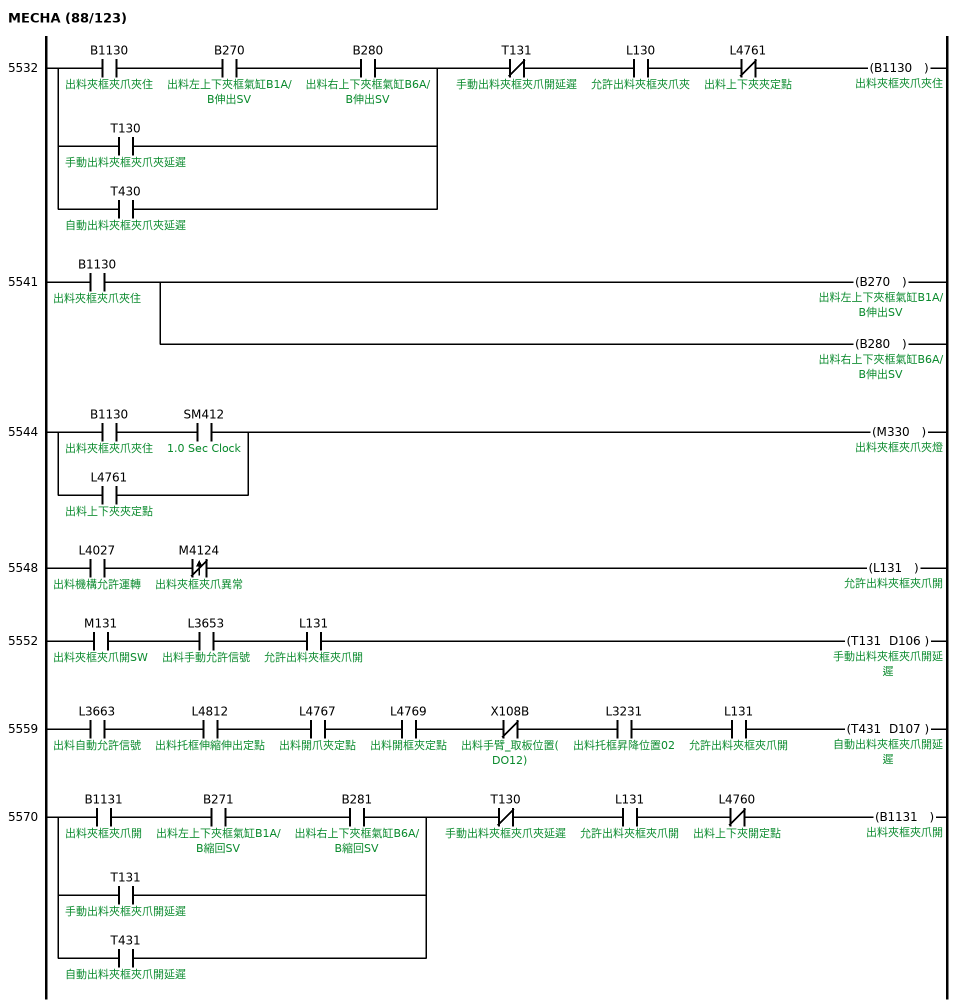
[picture p384: ladder of MECHA, rungs at steps 5532 to 5570]
5532  LD      B1130  ; 出料夾框夾爪夾住
      AND     B270  ; 出料左上下夾框氣缸B1A/B伸出SV
      AND     B280  ; 出料右上下夾框氣缸B6A/B伸出SV
      OR      T130  ; 手動出料夾框夾爪夾延遲
      OR      T430  ; 自動出料夾框夾爪夾延遲
      ANI     T131  ; 手動出料夾框夾爪開延遲
      AND     L130  ; 允許出料夾框夾爪夾
      ANI     L4761  ; 出料上下夾夾定點
      OUT     B1130  ; 出料夾框夾爪夾住
5541  LD      B1130  ; 出料夾框夾爪夾住
      OUT     B270  ; 出料左上下夾框氣缸B1A/B伸出SV
      OUT     B280  ; 出料右上下夾框氣缸B6A/B伸出SV
5544  LD      B1130  ; 出料夾框夾爪夾住
      AND     SM412  ; 1.0 Sec Clock
      OR      L4761  ; 出料上下夾夾定點
      OUT     M330  ; 出料夾框夾爪夾燈
5548  LD      L4027  ; 出料機構允許運轉
      ANDPI   M4124  ; 出料夾框夾爪異常
      OUT     L131  ; 允許出料夾框夾爪開
5552  LD      M131  ; 出料夾框夾爪開SW
      AND     L3653  ; 出料手動允許信號
      AND     L131  ; 允許出料夾框夾爪開
      OUT     T131 D106  ; 手動出料夾框夾爪開延遲
5559  LD      L3663  ; 出料自動允許信號
      AND     L4812  ; 出料托框伸縮伸出定點
      AND     L4767  ; 出料開爪夾定點
      AND     L4769  ; 出料開框夾定點
      ANI     X108B  ; 出料手臂_取板位置(DO12)
      AND     L3231  ; 出料托框昇降位置02
      AND     L131  ; 允許出料夾框夾爪開
      OUT     T431 D107  ; 自動出料夾框夾爪開延遲
5570  LD      B1131  ; 出料夾框夾爪開
      AND     B271  ; 出料左上下夾框氣缸B1A/B縮回SV
      AND     B281  ; 出料右上下夾框氣缸B6A/B縮回SV
      OR      T131  ; 手動出料夾框夾爪開延遲
      OR      T431  ; 自動出料夾框夾爪開延遲
      ANI     T130  ; 手動出料夾框夾爪夾延遲
      AND     L131  ; 允許出料夾框夾爪開
      ANI     L4760  ; 出料上下夾開定點
      OUT     B1131  ; 出料夾框夾爪開
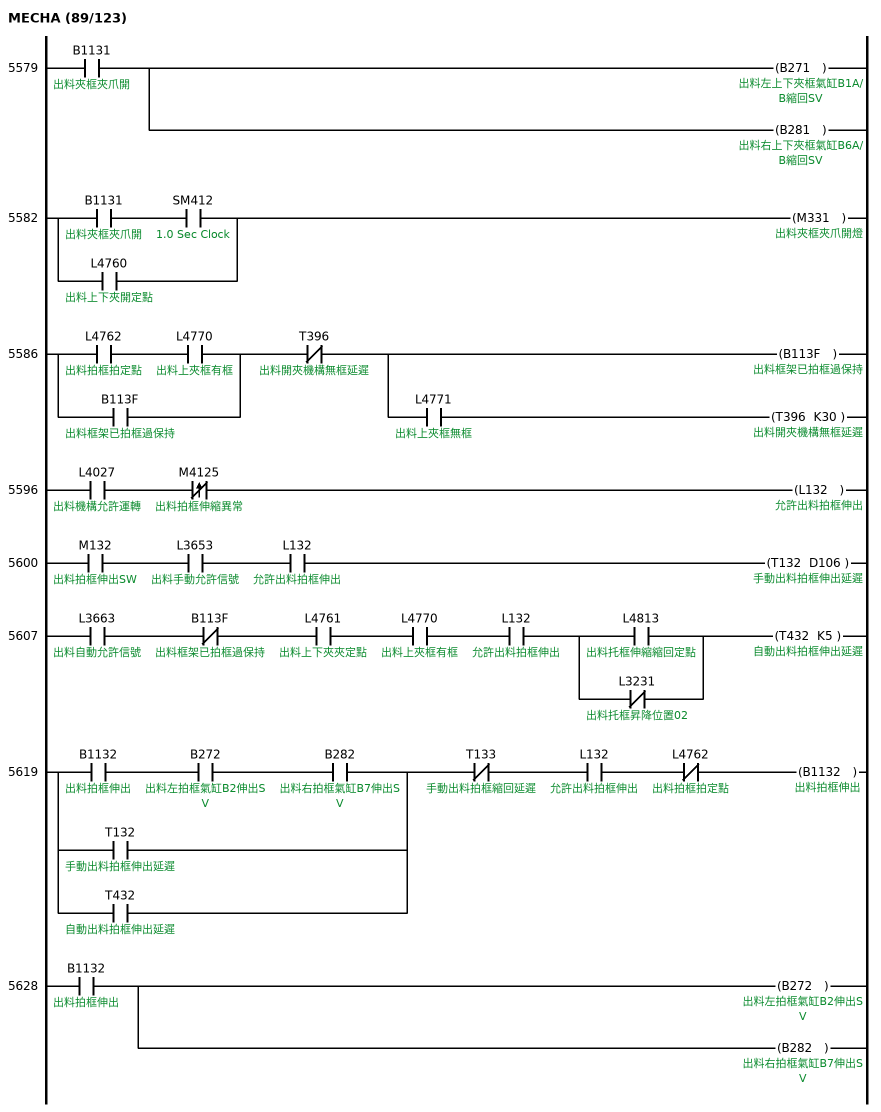
5579  LD      B1131  ; 出料夾框夾爪開
      OUT     B271  ; 出料左上下夾框氣缸B1A/B縮回SV
      OUT     B281  ; 出料右上下夾框氣缸B6A/B縮回SV
5582  LD      B1131  ; 出料夾框夾爪開
      AND     SM412  ; 1.0 Sec Clock
      OR      L4760  ; 出料上下夾開定點
      OUT     M331  ; 出料夾框夾爪開燈
5586  LD      L4762  ; 出料拍框拍定點
      AND     L4770  ; 出料上夾框有框
      OR      B113F  ; 出料框架已拍框過保持
      ANI     T396  ; 出料開夾機構無框延遲
      OUT     B113F  ; 出料框架已拍框過保持
      AND     L4771  ; 出料上夾框無框
      OUT     T396 K30  ; 出料開夾機構無框延遲
5596  LD      L4027  ; 出料機構允許運轉
      ANDPI   M4125  ; 出料拍框伸縮異常
      OUT     L132  ; 允許出料拍框伸出
5600  LD      M132  ; 出料拍框伸出SW
      AND     L3653  ; 出料手動允許信號
      AND     L132  ; 允許出料拍框伸出
      OUT     T132 D106  ; 手動出料拍框伸出延遲
5607  LD      L3663  ; 出料自動允許信號
      ANI     B113F  ; 出料框架已拍框過保持
      AND     L4761  ; 出料上下夾夾定點
      AND     L4770  ; 出料上夾框有框
      AND     L132  ; 允許出料拍框伸出
      LD      L4813  ; 出料托框伸縮縮回定點
      ORI     L3231  ; 出料托框昇降位置02
      ANB
      OUT     T432 K5  ; 自動出料拍框伸出延遲
5619  LD      B1132  ; 出料拍框伸出
      AND     B272  ; 出料左拍框氣缸B2伸出SV
      AND     B282  ; 出料右拍框氣缸B7伸出SV
      OR      T132  ; 手動出料拍框伸出延遲
      OR      T432  ; 自動出料拍框伸出延遲
      ANI     T133  ; 手動出料拍框縮回延遲
      AND     L132  ; 允許出料拍框伸出
      ANI     L4762  ; 出料拍框拍定點
      OUT     B1132  ; 出料拍框伸出
5628  LD      B1132  ; 出料拍框伸出
      OUT     B272  ; 出料左拍框氣缸B2伸出SV
      OUT     B282  ; 出料右拍框氣缸B7伸出SV
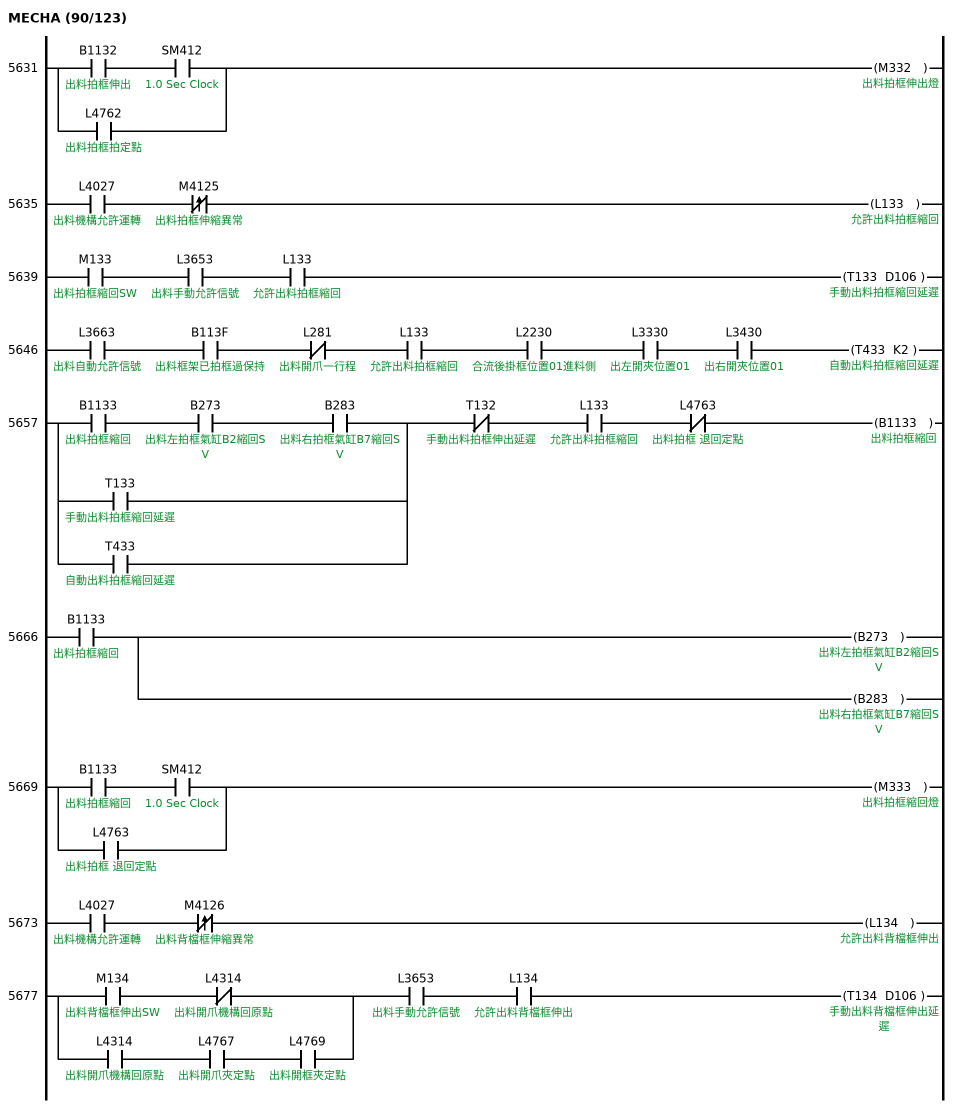
5631  LD      B1132  ; 出料拍框伸出
      AND     SM412  ; 1.0 Sec Clock
      OR      L4762  ; 出料拍框拍定點
      OUT     M332  ; 出料拍框伸出燈
5635  LD      L4027  ; 出料機構允許運轉
      ANDPI   M4125  ; 出料拍框伸縮異常
      OUT     L133  ; 允許出料拍框縮回
5639  LD      M133  ; 出料拍框縮回SW
      AND     L3653  ; 出料手動允許信號
      AND     L133  ; 允許出料拍框縮回
      OUT     T133 D106  ; 手動出料拍框縮回延遲
5646  LD      L3663  ; 出料自動允許信號
      AND     B113F  ; 出料框架已拍框過保持
      ANI     L281  ; 出料開爪一行程
      AND     L133  ; 允許出料拍框縮回
      AND     L2230  ; 合流後掛框位置01進料側
      AND     L3330  ; 出左開夾位置01
      AND     L3430  ; 出右開夾位置01
      OUT     T433 K2  ; 自動出料拍框縮回延遲
5657  LD      B1133  ; 出料拍框縮回
      AND     B273  ; 出料左拍框氣缸B2縮回SV
      AND     B283  ; 出料右拍框氣缸B7縮回SV
      OR      T133  ; 手動出料拍框縮回延遲
      OR      T433  ; 自動出料拍框縮回延遲
      ANI     T132  ; 手動出料拍框伸出延遲
      AND     L133  ; 允許出料拍框縮回
      ANI     L4763  ; 出料拍框 退回定點
      OUT     B1133  ; 出料拍框縮回
5666  LD      B1133  ; 出料拍框縮回
      OUT     B273  ; 出料左拍框氣缸B2縮回SV
      OUT     B283  ; 出料右拍框氣缸B7縮回SV
5669  LD      B1133  ; 出料拍框縮回
      AND     SM412  ; 1.0 Sec Clock
      OR      L4763  ; 出料拍框 退回定點
      OUT     M333  ; 出料拍框縮回燈
5673  LD      L4027  ; 出料機構允許運轉
      ANDPI   M4126  ; 出料背檔框伸縮異常
      OUT     L134  ; 允許出料背檔框伸出
5677  LD      M134  ; 出料背檔框伸出SW
      ANI     L4314  ; 出料開爪機構回原點
      LD      L4314  ; 出料開爪機構回原點
      AND     L4767  ; 出料開爪夾定點
      AND     L4769  ; 出料開框夾定點
      ORB
      AND     L3653  ; 出料手動允許信號
      AND     L134  ; 允許出料背檔框伸出
      OUT     T134 D106  ; 手動出料背檔框伸出延遲
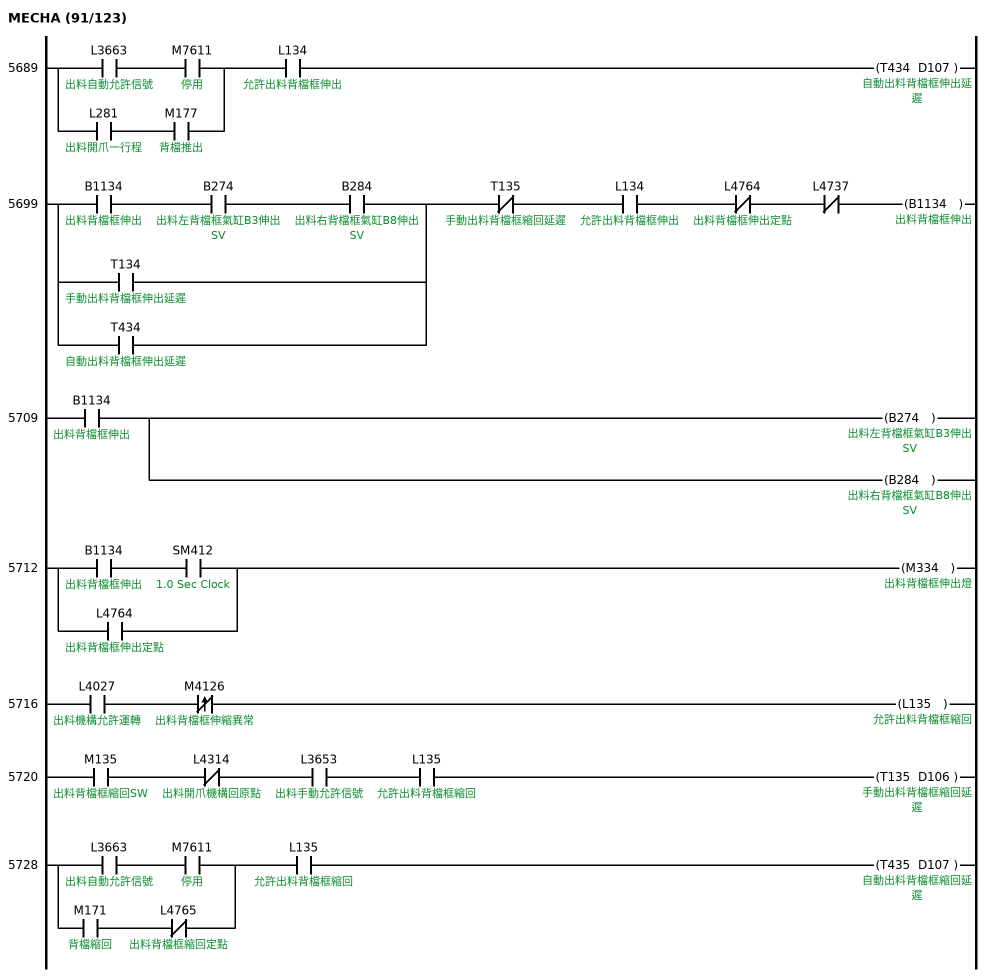
5689  LD      L3663  ; 出料自動允許信號
      AND     M7611  ; 停用
      LD      L281  ; 出料開爪一行程
      AND     M177  ; 背檔推出
      ORB
      AND     L134  ; 允許出料背檔框伸出
      OUT     T434 D107  ; 自動出料背檔框伸出延遲
5699  LD      B1134  ; 出料背檔框伸出
      AND     B274  ; 出料左背檔框氣缸B3伸出SV
      AND     B284  ; 出料右背檔框氣缸B8伸出SV
      OR      T134  ; 手動出料背檔框伸出延遲
      OR      T434  ; 自動出料背檔框伸出延遲
      ANI     T135  ; 手動出料背檔框縮回延遲
      AND     L134  ; 允許出料背檔框伸出
      ANI     L4764  ; 出料背檔框伸出定點
      ANI     L4737
      OUT     B1134  ; 出料背檔框伸出
5709  LD      B1134  ; 出料背檔框伸出
      OUT     B274  ; 出料左背檔框氣缸B3伸出SV
      OUT     B284  ; 出料右背檔框氣缸B8伸出SV
5712  LD      B1134  ; 出料背檔框伸出
      AND     SM412  ; 1.0 Sec Clock
      OR      L4764  ; 出料背檔框伸出定點
      OUT     M334  ; 出料背檔框伸出燈
5716  LD      L4027  ; 出料機構允許運轉
      ANDPI   M4126  ; 出料背檔框伸縮異常
      OUT     L135  ; 允許出料背檔框縮回
5720  LD      M135  ; 出料背檔框縮回SW
      ANI     L4314  ; 出料開爪機構回原點
      AND     L3653  ; 出料手動允許信號
      AND     L135  ; 允許出料背檔框縮回
      OUT     T135 D106  ; 手動出料背檔框縮回延遲
5728  LD      L3663  ; 出料自動允許信號
      AND     M7611  ; 停用
      LD      M171  ; 背檔縮回
      ANI     L4765  ; 出料背檔框縮回定點
      ORB
      AND     L135  ; 允許出料背檔框縮回
      OUT     T435 D107  ; 自動出料背檔框縮回延遲
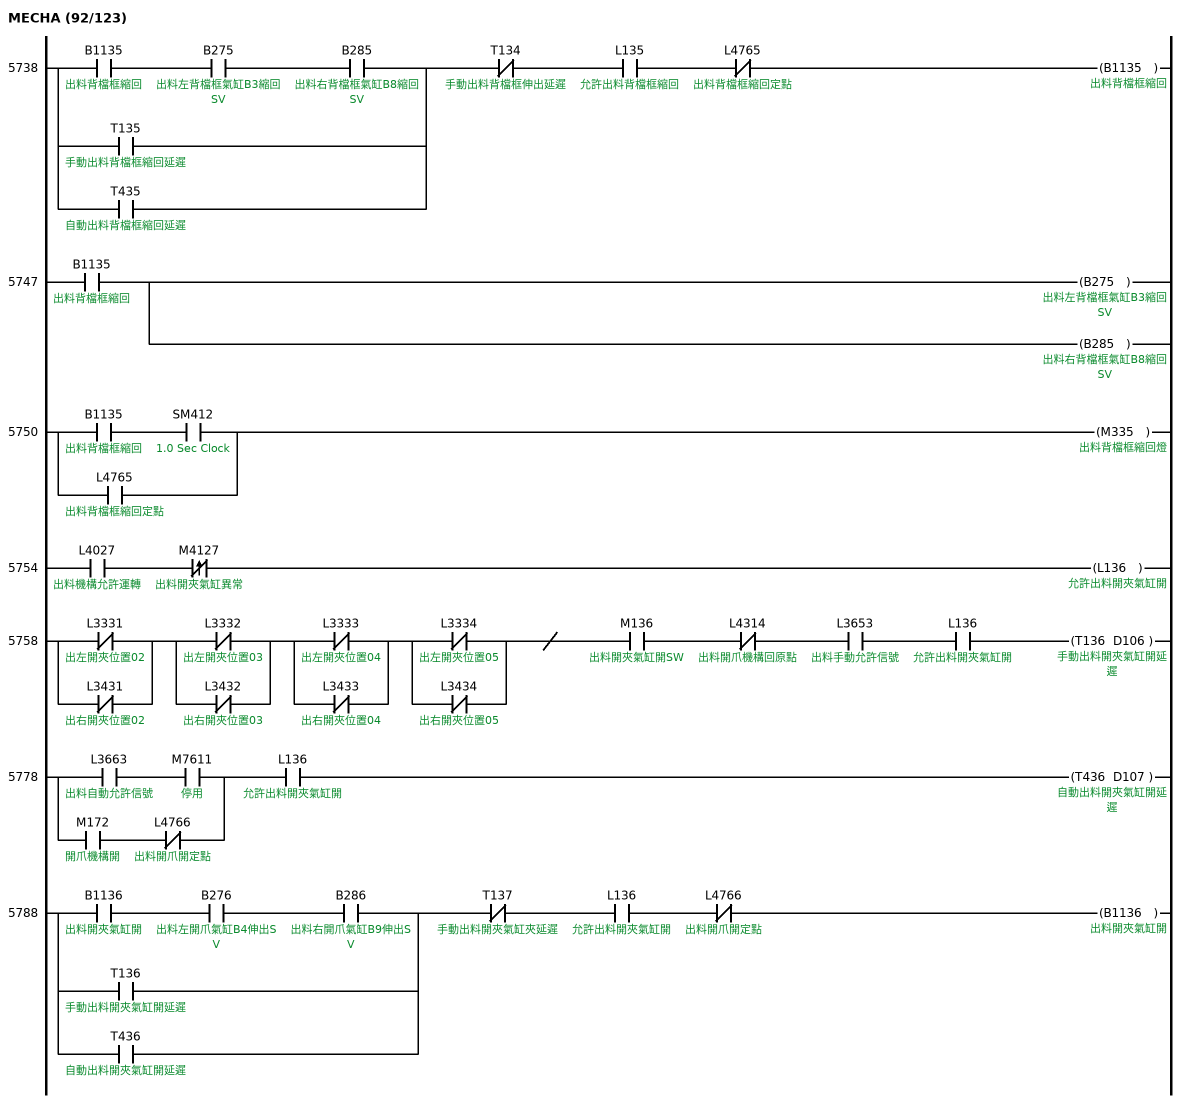
5738  LD      B1135  ; 出料背檔框縮回
      AND     B275  ; 出料左背檔框氣缸B3縮回SV
      AND     B285  ; 出料右背檔框氣缸B8縮回SV
      OR      T135  ; 手動出料背檔框縮回延遲
      OR      T435  ; 自動出料背檔框縮回延遲
      ANI     T134  ; 手動出料背檔框伸出延遲
      AND     L135  ; 允許出料背檔框縮回
      ANI     L4765  ; 出料背檔框縮回定點
      OUT     B1135  ; 出料背檔框縮回
5747  LD      B1135  ; 出料背檔框縮回
      OUT     B275  ; 出料左背檔框氣缸B3縮回SV
      OUT     B285  ; 出料右背檔框氣缸B8縮回SV
5750  LD      B1135  ; 出料背檔框縮回
      AND     SM412  ; 1.0 Sec Clock
      OR      L4765  ; 出料背檔框縮回定點
      OUT     M335  ; 出料背檔框縮回燈
5754  LD      L4027  ; 出料機構允許運轉
      ANDPI   M4127  ; 出料開夾氣缸異常
      OUT     L136  ; 允許出料開夾氣缸開
5758  LDI     L3331  ; 出左開夾位置02
      ORI     L3431  ; 出右開夾位置02
      LDI     L3332  ; 出左開夾位置03
      ORI     L3432  ; 出右開夾位置03
      ANB
      LDI     L3333  ; 出左開夾位置04
      ORI     L3433  ; 出右開夾位置04
      ANB
      LDI     L3334  ; 出左開夾位置05
      ORI     L3434  ; 出右開夾位置05
      ANB
      INV
      AND     M136  ; 出料開夾氣缸開SW
      ANI     L4314  ; 出料開爪機構回原點
      AND     L3653  ; 出料手動允許信號
      AND     L136  ; 允許出料開夾氣缸開
      OUT     T136 D106  ; 手動出料開夾氣缸開延遲
5778  LD      L3663  ; 出料自動允許信號
      AND     M7611  ; 停用
      LD      M172  ; 開爪機構開
      ANI     L4766  ; 出料開爪開定點
      ORB
      AND     L136  ; 允許出料開夾氣缸開
      OUT     T436 D107  ; 自動出料開夾氣缸開延遲
5788  LD      B1136  ; 出料開夾氣缸開
      AND     B276  ; 出料左開爪氣缸B4伸出SV
      AND     B286  ; 出料右開爪氣缸B9伸出SV
      OR      T136  ; 手動出料開夾氣缸開延遲
      OR      T436  ; 自動出料開夾氣缸開延遲
      ANI     T137  ; 手動出料開夾氣缸夾延遲
      AND     L136  ; 允許出料開夾氣缸開
      ANI     L4766  ; 出料開爪開定點
      OUT     B1136  ; 出料開夾氣缸開
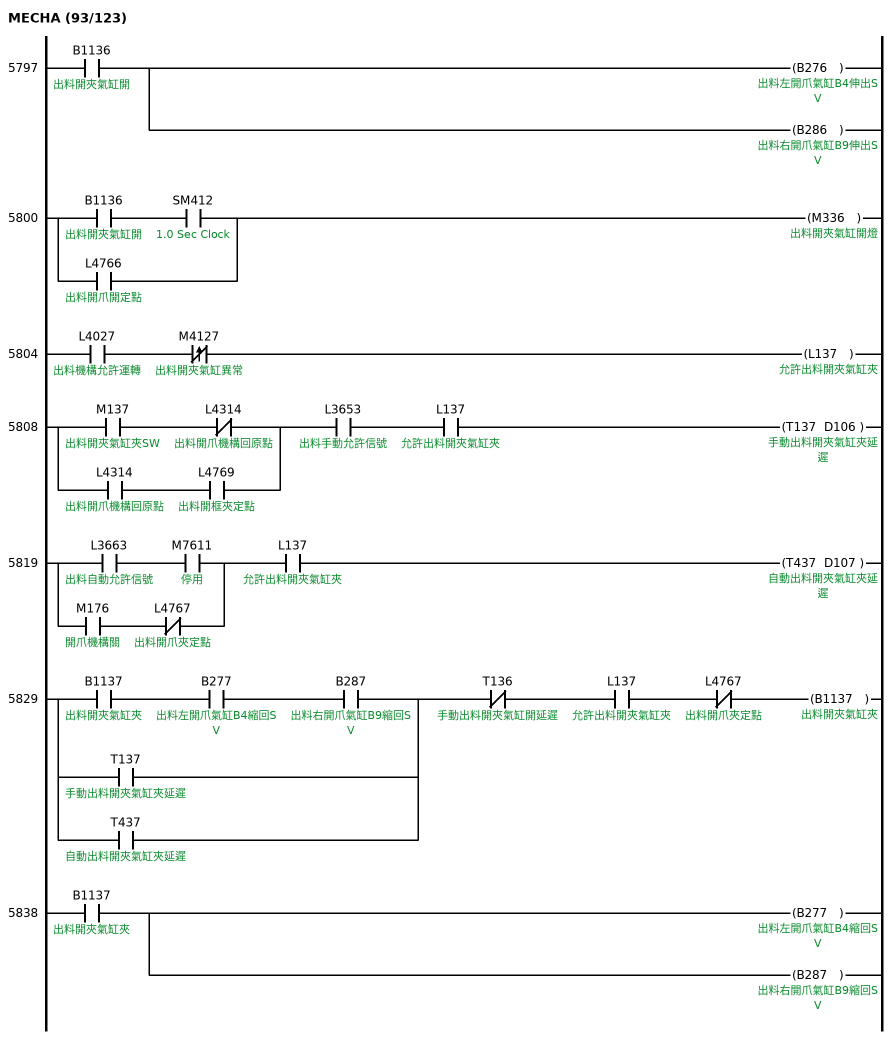
5797  LD      B1136  ; 出料開夾氣缸開
      OUT     B276  ; 出料左開爪氣缸B4伸出SV
      OUT     B286  ; 出料右開爪氣缸B9伸出SV
5800  LD      B1136  ; 出料開夾氣缸開
      AND     SM412  ; 1.0 Sec Clock
      OR      L4766  ; 出料開爪開定點
      OUT     M336  ; 出料開夾氣缸開燈
5804  LD      L4027  ; 出料機構允許運轉
      ANDPI   M4127  ; 出料開夾氣缸異常
      OUT     L137  ; 允許出料開夾氣缸夾
5808  LD      M137  ; 出料開夾氣缸夾SW
      ANI     L4314  ; 出料開爪機構回原點
      LD      L4314  ; 出料開爪機構回原點
      AND     L4769  ; 出料開框夾定點
      ORB
      AND     L3653  ; 出料手動允許信號
      AND     L137  ; 允許出料開夾氣缸夾
      OUT     T137 D106  ; 手動出料開夾氣缸夾延遲
5819  LD      L3663  ; 出料自動允許信號
      AND     M7611  ; 停用
      LD      M176  ; 開爪機構關
      ANI     L4767  ; 出料開爪夾定點
      ORB
      AND     L137  ; 允許出料開夾氣缸夾
      OUT     T437 D107  ; 自動出料開夾氣缸夾延遲
5829  LD      B1137  ; 出料開夾氣缸夾
      AND     B277  ; 出料左開爪氣缸B4縮回SV
      AND     B287  ; 出料右開爪氣缸B9縮回SV
      OR      T137  ; 手動出料開夾氣缸夾延遲
      OR      T437  ; 自動出料開夾氣缸夾延遲
      ANI     T136  ; 手動出料開夾氣缸開延遲
      AND     L137  ; 允許出料開夾氣缸夾
      ANI     L4767  ; 出料開爪夾定點
      OUT     B1137  ; 出料開夾氣缸夾
5838  LD      B1137  ; 出料開夾氣缸夾
      OUT     B277  ; 出料左開爪氣缸B4縮回SV
      OUT     B287  ; 出料右開爪氣缸B9縮回SV
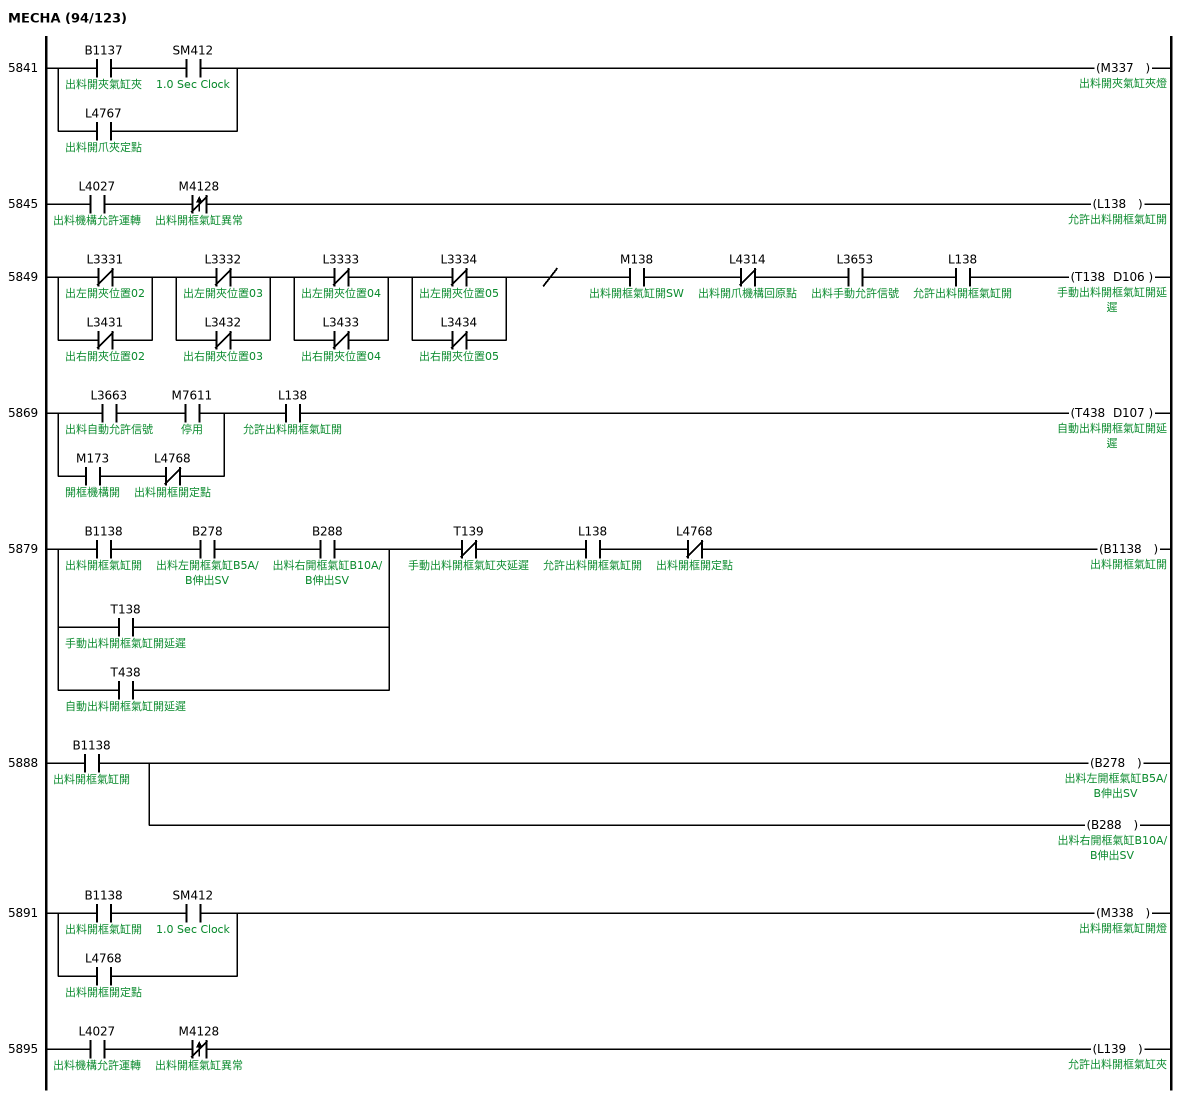
5841  LD      B1137  ; 出料開夾氣缸夾
      AND     SM412  ; 1.0 Sec Clock
      OR      L4767  ; 出料開爪夾定點
      OUT     M337  ; 出料開夾氣缸夾燈
5845  LD      L4027  ; 出料機構允許運轉
      ANDPI   M4128  ; 出料開框氣缸異常
      OUT     L138  ; 允許出料開框氣缸開
5849  LDI     L3331  ; 出左開夾位置02
      ORI     L3431  ; 出右開夾位置02
      LDI     L3332  ; 出左開夾位置03
      ORI     L3432  ; 出右開夾位置03
      ANB
      LDI     L3333  ; 出左開夾位置04
      ORI     L3433  ; 出右開夾位置04
      ANB
      LDI     L3334  ; 出左開夾位置05
      ORI     L3434  ; 出右開夾位置05
      ANB
      INV
      AND     M138  ; 出料開框氣缸開SW
      ANI     L4314  ; 出料開爪機構回原點
      AND     L3653  ; 出料手動允許信號
      AND     L138  ; 允許出料開框氣缸開
      OUT     T138 D106  ; 手動出料開框氣缸開延遲
5869  LD      L3663  ; 出料自動允許信號
      AND     M7611  ; 停用
      LD      M173  ; 開框機構開
      ANI     L4768  ; 出料開框開定點
      ORB
      AND     L138  ; 允許出料開框氣缸開
      OUT     T438 D107  ; 自動出料開框氣缸開延遲
5879  LD      B1138  ; 出料開框氣缸開
      AND     B278  ; 出料左開框氣缸B5A/B伸出SV
      AND     B288  ; 出料右開框氣缸B10A/B伸出SV
      OR      T138  ; 手動出料開框氣缸開延遲
      OR      T438  ; 自動出料開框氣缸開延遲
      ANI     T139  ; 手動出料開框氣缸夾延遲
      AND     L138  ; 允許出料開框氣缸開
      ANI     L4768  ; 出料開框開定點
      OUT     B1138  ; 出料開框氣缸開
5888  LD      B1138  ; 出料開框氣缸開
      OUT     B278  ; 出料左開框氣缸B5A/B伸出SV
      OUT     B288  ; 出料右開框氣缸B10A/B伸出SV
5891  LD      B1138  ; 出料開框氣缸開
      AND     SM412  ; 1.0 Sec Clock
      OR      L4768  ; 出料開框開定點
      OUT     M338  ; 出料開框氣缸開燈
5895  LD      L4027  ; 出料機構允許運轉
      ANDPI   M4128  ; 出料開框氣缸異常
      OUT     L139  ; 允許出料開框氣缸夾
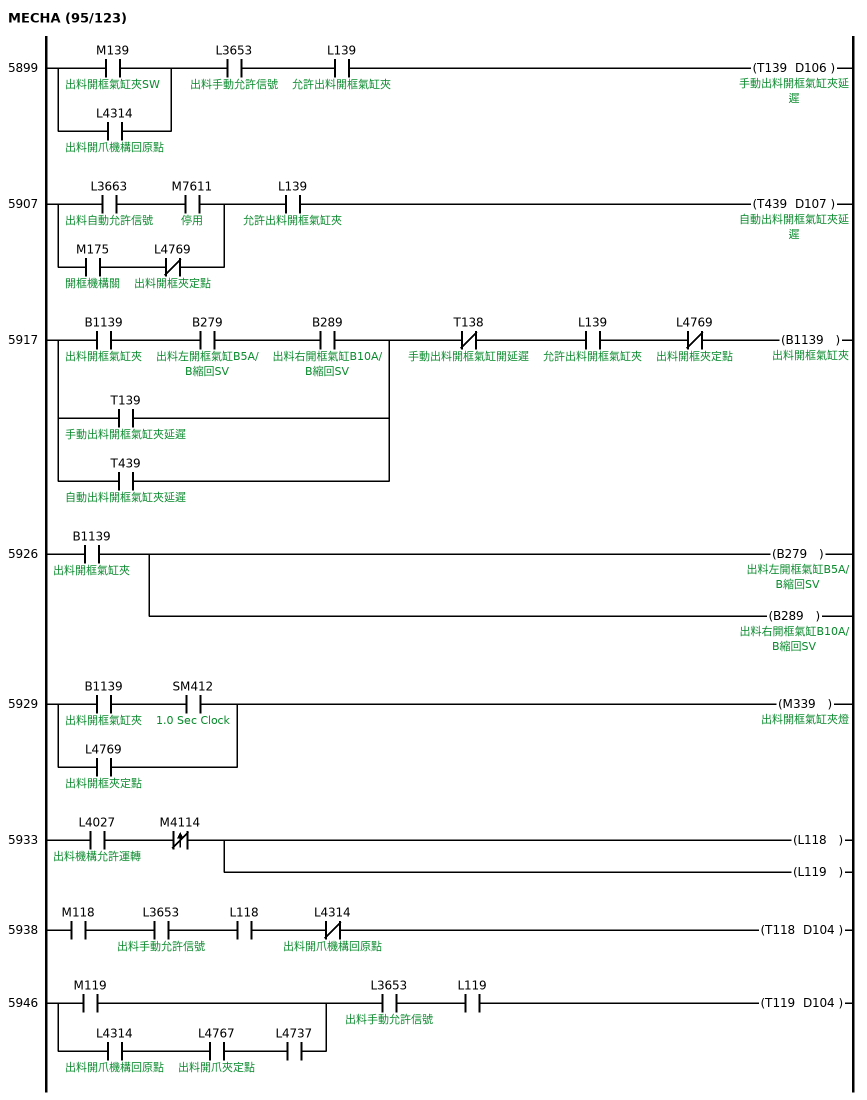
5899  LD      M139  ; 出料開框氣缸夾SW
      OR      L4314  ; 出料開爪機構回原點
      AND     L3653  ; 出料手動允許信號
      AND     L139  ; 允許出料開框氣缸夾
      OUT     T139 D106  ; 手動出料開框氣缸夾延遲
5907  LD      L3663  ; 出料自動允許信號
      AND     M7611  ; 停用
      LD      M175  ; 開框機構關
      ANI     L4769  ; 出料開框夾定點
      ORB
      AND     L139  ; 允許出料開框氣缸夾
      OUT     T439 D107  ; 自動出料開框氣缸夾延遲
5917  LD      B1139  ; 出料開框氣缸夾
      AND     B279  ; 出料左開框氣缸B5A/B縮回SV
      AND     B289  ; 出料右開框氣缸B10A/B縮回SV
      OR      T139  ; 手動出料開框氣缸夾延遲
      OR      T439  ; 自動出料開框氣缸夾延遲
      ANI     T138  ; 手動出料開框氣缸開延遲
      AND     L139  ; 允許出料開框氣缸夾
      ANI     L4769  ; 出料開框夾定點
      OUT     B1139  ; 出料開框氣缸夾
5926  LD      B1139  ; 出料開框氣缸夾
      OUT     B279  ; 出料左開框氣缸B5A/B縮回SV
      OUT     B289  ; 出料右開框氣缸B10A/B縮回SV
5929  LD      B1139  ; 出料開框氣缸夾
      AND     SM412  ; 1.0 Sec Clock
      OR      L4769  ; 出料開框夾定點
      OUT     M339  ; 出料開框氣缸夾燈
5933  LD      L4027  ; 出料機構允許運轉
      ANDPI   M4114
      OUT     L118
      OUT     L119
5938  LD      M118
      AND     L3653  ; 出料手動允許信號
      AND     L118
      ANI     L4314  ; 出料開爪機構回原點
      OUT     T118 D104
5946  LD      M119
      LD      L4314  ; 出料開爪機構回原點
      AND     L4767  ; 出料開爪夾定點
      AND     L4737
      ORB
      AND     L3653  ; 出料手動允許信號
      AND     L119
      OUT     T119 D104
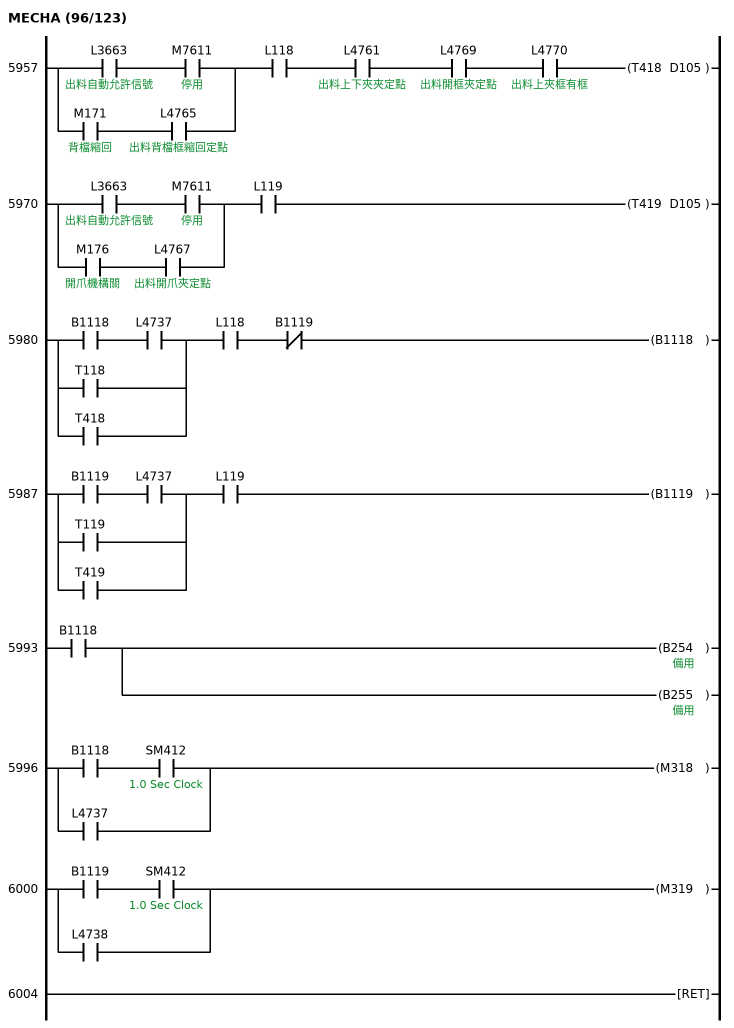
5957  LD      L3663  ; 出料自動允許信號
      AND     M7611  ; 停用
      LD      M171  ; 背檔縮回
      AND     L4765  ; 出料背檔框縮回定點
      ORB
      AND     L118
      AND     L4761  ; 出料上下夾夾定點
      AND     L4769  ; 出料開框夾定點
      AND     L4770  ; 出料上夾框有框
      OUT     T418 D105
5970  LD      L3663  ; 出料自動允許信號
      AND     M7611  ; 停用
      LD      M176  ; 開爪機構關
      AND     L4767  ; 出料開爪夾定點
      ORB
      AND     L119
      OUT     T419 D105
5980  LD      B1118
      AND     L4737
      OR      T118
      OR      T418
      AND     L118
      ANI     B1119
      OUT     B1118
5987  LD      B1119
      AND     L4737
      OR      T119
      OR      T419
      AND     L119
      OUT     B1119
5993  LD      B1118
      OUT     B254  ; 備用
      OUT     B255  ; 備用
5996  LD      B1118
      AND     SM412  ; 1.0 Sec Clock
      OR      L4737
      OUT     M318
6000  LD      B1119
      AND     SM412  ; 1.0 Sec Clock
      OR      L4738
      OUT     M319
6004  RET
      P1061
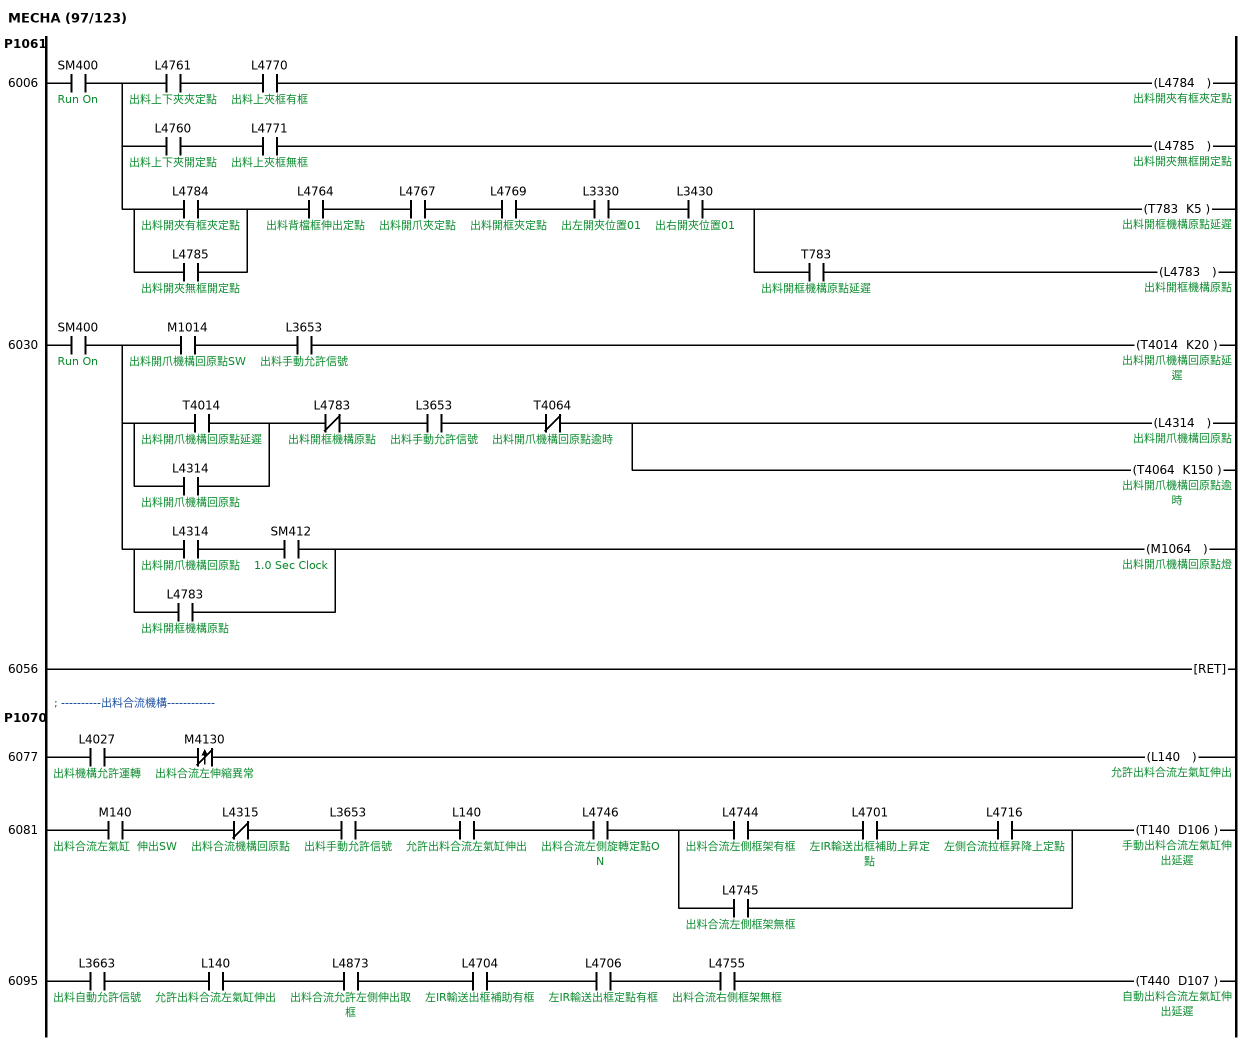
6006  LD      SM400  ; Run On
      MPS
      AND     L4761  ; 出料上下夾夾定點
      AND     L4770  ; 出料上夾框有框
      OUT     L4784  ; 出料開夾有框夾定點
      MRD
      AND     L4760  ; 出料上下夾開定點
      AND     L4771  ; 出料上夾框無框
      OUT     L4785  ; 出料開夾無框開定點
      MPP
      LD      L4784  ; 出料開夾有框夾定點
      OR      L4785  ; 出料開夾無框開定點
      ANB
      AND     L4764  ; 出料背檔框伸出定點
      AND     L4767  ; 出料開爪夾定點
      AND     L4769  ; 出料開框夾定點
      AND     L3330  ; 出左開夾位置01
      AND     L3430  ; 出右開夾位置01
      OUT     T783 K5  ; 出料開框機構原點延遲
      AND     T783  ; 出料開框機構原點延遲
      OUT     L4783  ; 出料開框機構原點
6030  LD      SM400  ; Run On
      MPS
      AND     M1014  ; 出料開爪機構回原點SW
      AND     L3653  ; 出料手動允許信號
      OUT     T4014 K20  ; 出料開爪機構回原點延遲
      MRD
      LD      T4014  ; 出料開爪機構回原點延遲
      OR      L4314  ; 出料開爪機構回原點
      ANB
      ANI     L4783  ; 出料開框機構原點
      AND     L3653  ; 出料手動允許信號
      ANI     T4064  ; 出料開爪機構回原點逾時
      OUT     L4314  ; 出料開爪機構回原點
      OUT     T4064 K150  ; 出料開爪機構回原點逾時
      MPP
      LD      L4314  ; 出料開爪機構回原點
      AND     SM412  ; 1.0 Sec Clock
      OR      L4783  ; 出料開框機構原點
      ANB
      OUT     M1064  ; 出料開爪機構回原點燈
6056  RET
; ----------出料合流機構------------
      P1070
6077  LD      L4027  ; 出料機構允許運轉
      ANDPI   M4130  ; 出料合流左伸縮異常
      OUT     L140  ; 允許出料合流左氣缸伸出
6081  LD      M140  ; 出料合流左氣缸  伸出SW
      ANI     L4315  ; 出料合流機構回原點
      AND     L3653  ; 出料手動允許信號
      AND     L140  ; 允許出料合流左氣缸伸出
      AND     L4746  ; 出料合流左側旋轉定點ON
      LD      L4744  ; 出料合流左側框架有框
      AND     L4701  ; 左IR輸送出框補助上昇定點
      AND     L4716  ; 左側合流拉框昇降上定點
      OR      L4745  ; 出料合流左側框架無框
      ANB
      OUT     T140 D106  ; 手動出料合流左氣缸伸出延遲
6095  LD      L3663  ; 出料自動允許信號
      AND     L140  ; 允許出料合流左氣缸伸出
      AND     L4873  ; 出料合流允許左側伸出取框
      AND     L4704  ; 左IR輸送出框補助有框
      AND     L4706  ; 左IR輸送出框定點有框
      AND     L4755  ; 出料合流右側框架無框
      OUT     T440 D107  ; 自動出料合流左氣缸伸出延遲
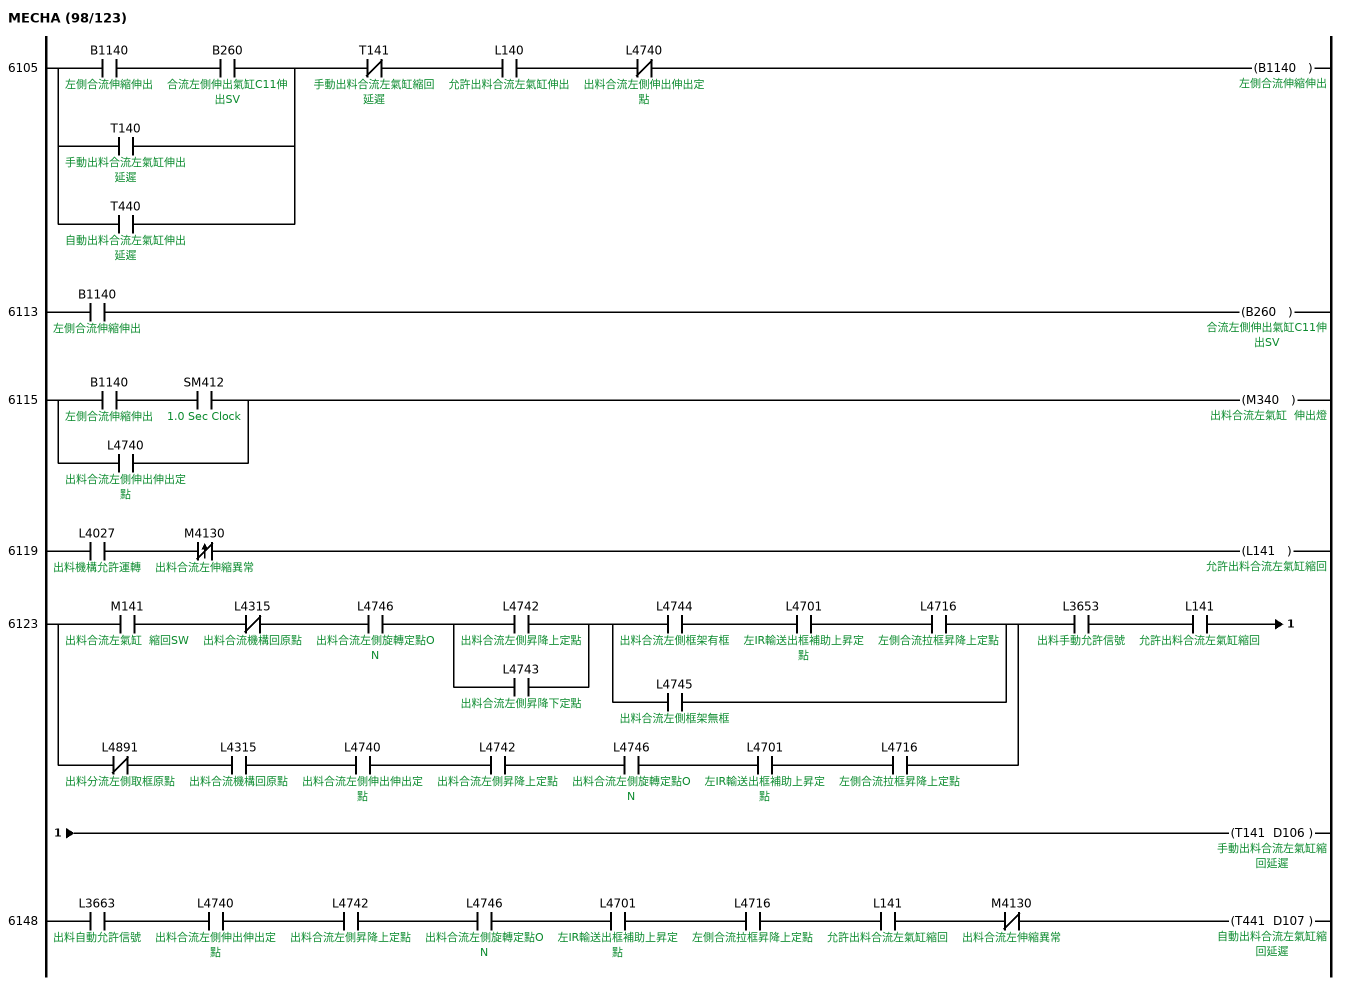
6105  LD      B1140  ; 左側合流伸縮伸出
      AND     B260  ; 合流左側伸出氣缸C11伸出SV
      OR      T140  ; 手動出料合流左氣缸伸出延遲
      OR      T440  ; 自動出料合流左氣缸伸出延遲
      ANI     T141  ; 手動出料合流左氣缸縮回延遲
      AND     L140  ; 允許出料合流左氣缸伸出
      ANI     L4740  ; 出料合流左側伸出伸出定點
      OUT     B1140  ; 左側合流伸縮伸出
6113  LD      B1140  ; 左側合流伸縮伸出
      OUT     B260  ; 合流左側伸出氣缸C11伸出SV
6115  LD      B1140  ; 左側合流伸縮伸出
      AND     SM412  ; 1.0 Sec Clock
      OR      L4740  ; 出料合流左側伸出伸出定點
      OUT     M340  ; 出料合流左氣缸  伸出燈
6119  LD      L4027  ; 出料機構允許運轉
      ANDPI   M4130  ; 出料合流左伸縮異常
      OUT     L141  ; 允許出料合流左氣缸縮回
6123  LD      M141  ; 出料合流左氣缸  縮回SW
      ANI     L4315  ; 出料合流機構回原點
      AND     L4746  ; 出料合流左側旋轉定點ON
      LD      L4742  ; 出料合流左側昇降上定點
      OR      L4743  ; 出料合流左側昇降下定點
      ANB
      LD      L4744  ; 出料合流左側框架有框
      AND     L4701  ; 左IR輸送出框補助上昇定點
      AND     L4716  ; 左側合流拉框昇降上定點
      OR      L4745  ; 出料合流左側框架無框
      ANB
      LDI     L4891  ; 出料分流左側取框原點
      AND     L4315  ; 出料合流機構回原點
      AND     L4740  ; 出料合流左側伸出伸出定點
      AND     L4742  ; 出料合流左側昇降上定點
      AND     L4746  ; 出料合流左側旋轉定點ON
      AND     L4701  ; 左IR輸送出框補助上昇定點
      AND     L4716  ; 左側合流拉框昇降上定點
      ORB
      AND     L3653  ; 出料手動允許信號
      AND     L141  ; 允許出料合流左氣缸縮回
      OUT     T141 D106  ; 手動出料合流左氣缸縮回延遲
6148  LD      L3663  ; 出料自動允許信號
      AND     L4740  ; 出料合流左側伸出伸出定點
      AND     L4742  ; 出料合流左側昇降上定點
      AND     L4746  ; 出料合流左側旋轉定點ON
      AND     L4701  ; 左IR輸送出框補助上昇定點
      AND     L4716  ; 左側合流拉框昇降上定點
      AND     L141  ; 允許出料合流左氣缸縮回
      ANI     M4130  ; 出料合流左伸縮異常
      OUT     T441 D107  ; 自動出料合流左氣缸縮回延遲
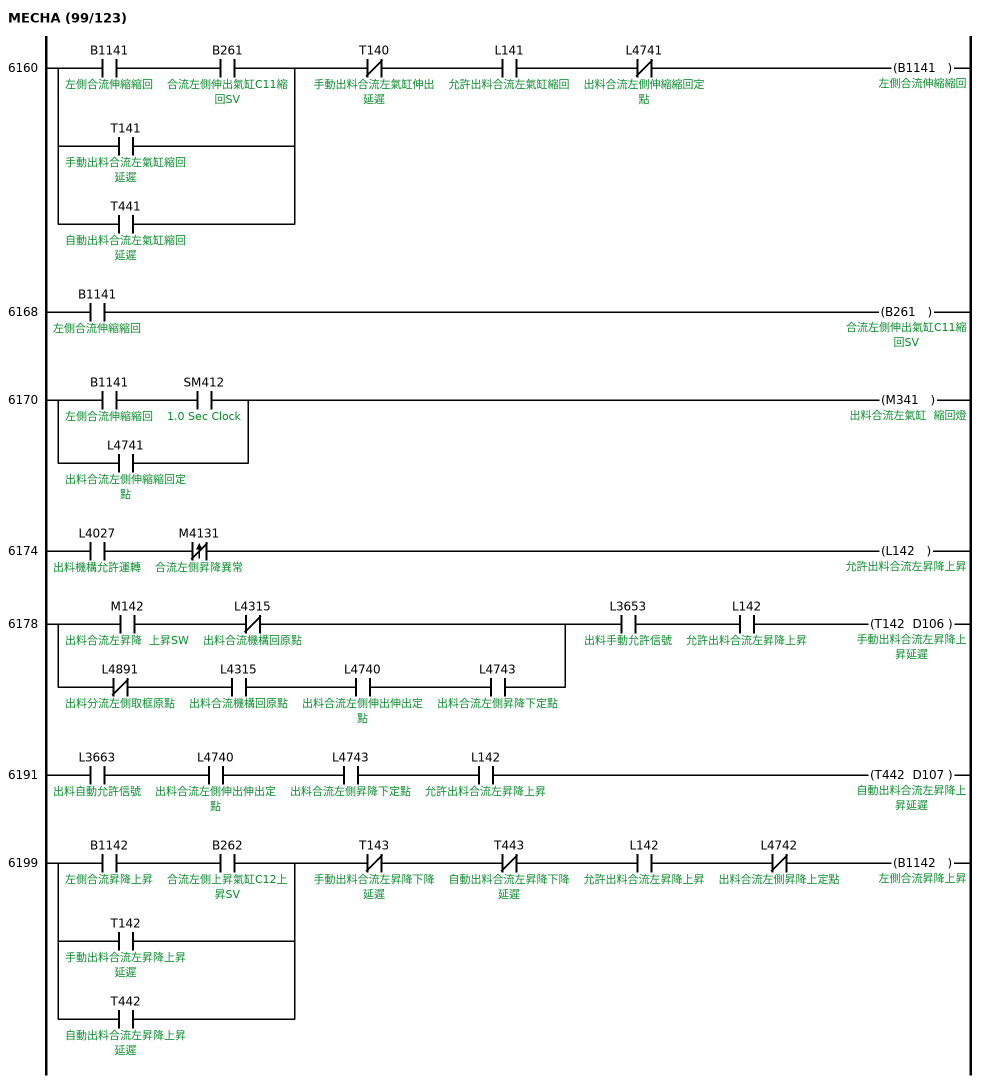
6160  LD      B1141  ; 左側合流伸縮縮回
      AND     B261  ; 合流左側伸出氣缸C11縮回SV
      OR      T141  ; 手動出料合流左氣缸縮回延遲
      OR      T441  ; 自動出料合流左氣缸縮回延遲
      ANI     T140  ; 手動出料合流左氣缸伸出延遲
      AND     L141  ; 允許出料合流左氣缸縮回
      ANI     L4741  ; 出料合流左側伸縮縮回定點
      OUT     B1141  ; 左側合流伸縮縮回
6168  LD      B1141  ; 左側合流伸縮縮回
      OUT     B261  ; 合流左側伸出氣缸C11縮回SV
6170  LD      B1141  ; 左側合流伸縮縮回
      AND     SM412  ; 1.0 Sec Clock
      OR      L4741  ; 出料合流左側伸縮縮回定點
      OUT     M341  ; 出料合流左氣缸  縮回燈
6174  LD      L4027  ; 出料機構允許運轉
      ANDPI   M4131  ; 合流左側昇降異常
      OUT     L142  ; 允許出料合流左昇降上昇
6178  LD      M142  ; 出料合流左昇降  上昇SW
      ANI     L4315  ; 出料合流機構回原點
      LDI     L4891  ; 出料分流左側取框原點
      AND     L4315  ; 出料合流機構回原點
      AND     L4740  ; 出料合流左側伸出伸出定點
      AND     L4743  ; 出料合流左側昇降下定點
      ORB
      AND     L3653  ; 出料手動允許信號
      AND     L142  ; 允許出料合流左昇降上昇
      OUT     T142 D106  ; 手動出料合流左昇降上昇延遲
6191  LD      L3663  ; 出料自動允許信號
      AND     L4740  ; 出料合流左側伸出伸出定點
      AND     L4743  ; 出料合流左側昇降下定點
      AND     L142  ; 允許出料合流左昇降上昇
      OUT     T442 D107  ; 自動出料合流左昇降上昇延遲
6199  LD      B1142  ; 左側合流昇降上昇
      AND     B262  ; 合流左側上昇氣缸C12上昇SV
      OR      T142  ; 手動出料合流左昇降上昇延遲
      OR      T442  ; 自動出料合流左昇降上昇延遲
      ANI     T143  ; 手動出料合流左昇降下降延遲
      ANI     T443  ; 自動出料合流左昇降下降延遲
      AND     L142  ; 允許出料合流左昇降上昇
      ANI     L4742  ; 出料合流左側昇降上定點
      OUT     B1142  ; 左側合流昇降上昇
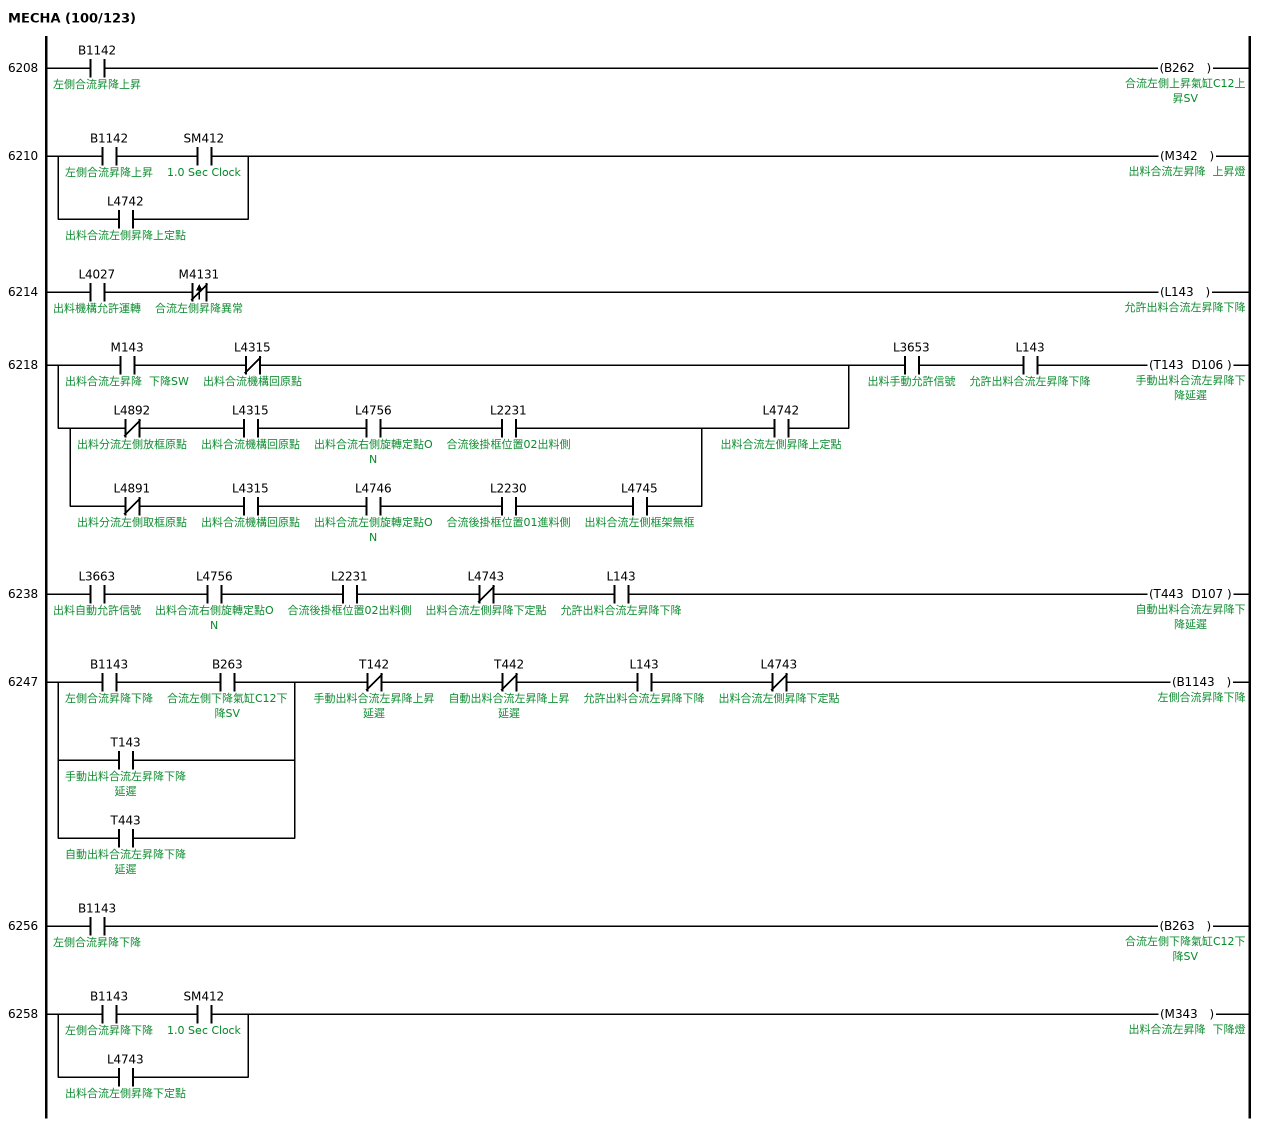
6208  LD      B1142  ; 左側合流昇降上昇
      OUT     B262  ; 合流左側上昇氣缸C12上昇SV
6210  LD      B1142  ; 左側合流昇降上昇
      AND     SM412  ; 1.0 Sec Clock
      OR      L4742  ; 出料合流左側昇降上定點
      OUT     M342  ; 出料合流左昇降  上昇燈
6214  LD      L4027  ; 出料機構允許運轉
      ANDPI   M4131  ; 合流左側昇降異常
      OUT     L143  ; 允許出料合流左昇降下降
6218  LD      M143  ; 出料合流左昇降  下降SW
      ANI     L4315  ; 出料合流機構回原點
      LDI     L4892  ; 出料分流左側放框原點
      AND     L4315  ; 出料合流機構回原點
      AND     L4756  ; 出料合流右側旋轉定點ON
      AND     L2231  ; 合流後掛框位置02出料側
      LDI     L4891  ; 出料分流左側取框原點
      AND     L4315  ; 出料合流機構回原點
      AND     L4746  ; 出料合流左側旋轉定點ON
      AND     L2230  ; 合流後掛框位置01進料側
      AND     L4745  ; 出料合流左側框架無框
      ORB
      AND     L4742  ; 出料合流左側昇降上定點
      ORB
      AND     L3653  ; 出料手動允許信號
      AND     L143  ; 允許出料合流左昇降下降
      OUT     T143 D106  ; 手動出料合流左昇降下降延遲
6238  LD      L3663  ; 出料自動允許信號
      AND     L4756  ; 出料合流右側旋轉定點ON
      AND     L2231  ; 合流後掛框位置02出料側
      ANI     L4743  ; 出料合流左側昇降下定點
      AND     L143  ; 允許出料合流左昇降下降
      OUT     T443 D107  ; 自動出料合流左昇降下降延遲
6247  LD      B1143  ; 左側合流昇降下降
      AND     B263  ; 合流左側下降氣缸C12下降SV
      OR      T143  ; 手動出料合流左昇降下降延遲
      OR      T443  ; 自動出料合流左昇降下降延遲
      ANI     T142  ; 手動出料合流左昇降上昇延遲
      ANI     T442  ; 自動出料合流左昇降上昇延遲
      AND     L143  ; 允許出料合流左昇降下降
      ANI     L4743  ; 出料合流左側昇降下定點
      OUT     B1143  ; 左側合流昇降下降
6256  LD      B1143  ; 左側合流昇降下降
      OUT     B263  ; 合流左側下降氣缸C12下降SV
6258  LD      B1143  ; 左側合流昇降下降
      AND     SM412  ; 1.0 Sec Clock
      OR      L4743  ; 出料合流左側昇降下定點
      OUT     M343  ; 出料合流左昇降  下降燈
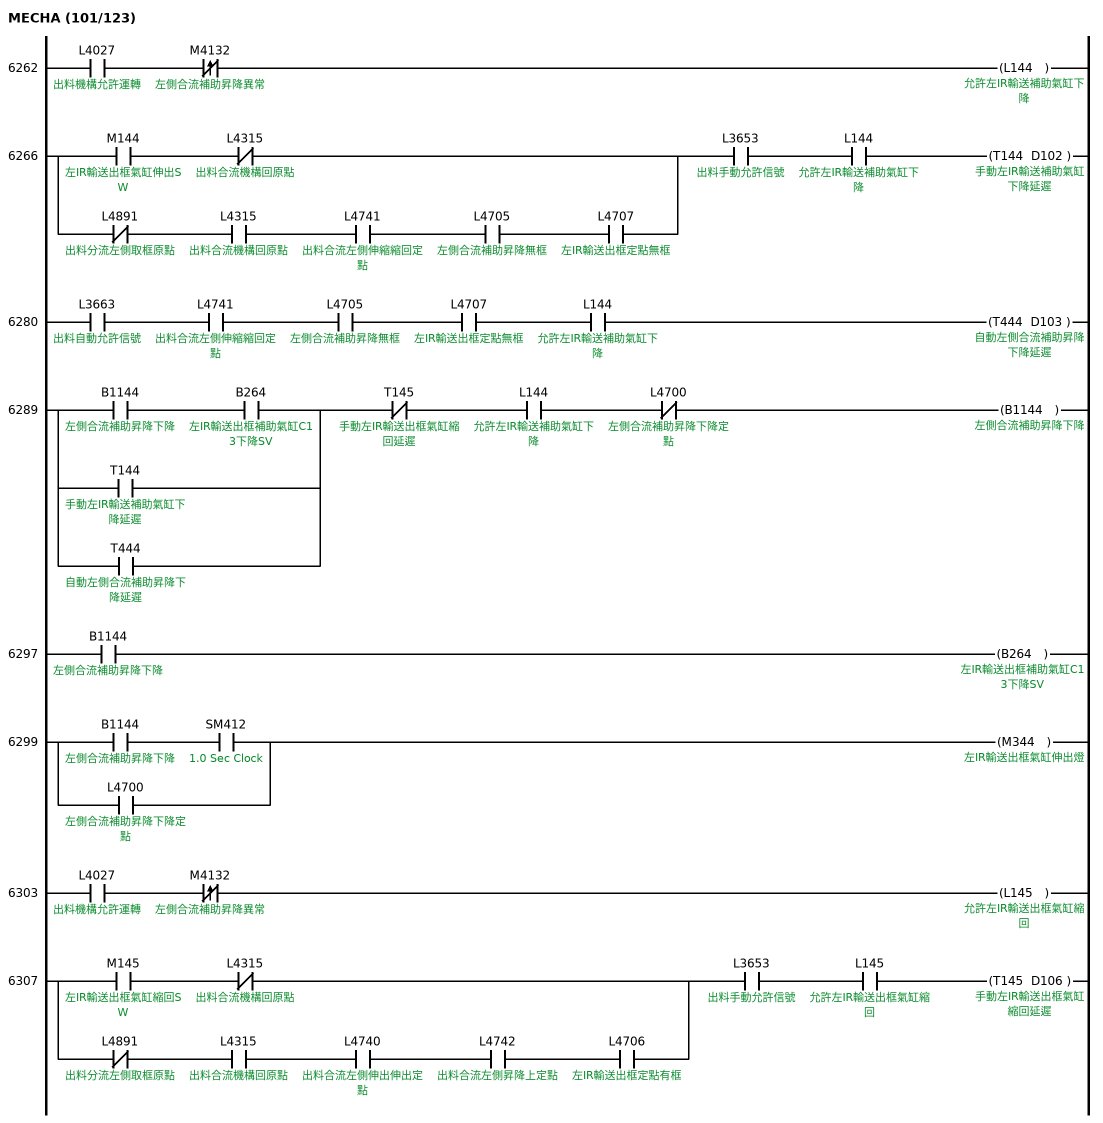
6262  LD      L4027  ; 出料機構允許運轉
      ANDPI   M4132  ; 左側合流補助昇降異常
      OUT     L144  ; 允許左IR輸送補助氣缸下降
6266  LD      M144  ; 左IR輸送出框氣缸伸出SW
      ANI     L4315  ; 出料合流機構回原點
      LDI     L4891  ; 出料分流左側取框原點
      AND     L4315  ; 出料合流機構回原點
      AND     L4741  ; 出料合流左側伸縮縮回定點
      AND     L4705  ; 左側合流補助昇降無框
      AND     L4707  ; 左IR輸送出框定點無框
      ORB
      AND     L3653  ; 出料手動允許信號
      AND     L144  ; 允許左IR輸送補助氣缸下降
      OUT     T144 D102  ; 手動左IR輸送補助氣缸下降延遲
6280  LD      L3663  ; 出料自動允許信號
      AND     L4741  ; 出料合流左側伸縮縮回定點
      AND     L4705  ; 左側合流補助昇降無框
      AND     L4707  ; 左IR輸送出框定點無框
      AND     L144  ; 允許左IR輸送補助氣缸下降
      OUT     T444 D103  ; 自動左側合流補助昇降下降延遲
6289  LD      B1144  ; 左側合流補助昇降下降
      AND     B264  ; 左IR輸送出框補助氣缸C13下降SV
      OR      T144  ; 手動左IR輸送補助氣缸下降延遲
      OR      T444  ; 自動左側合流補助昇降下降延遲
      ANI     T145  ; 手動左IR輸送出框氣缸縮回延遲
      AND     L144  ; 允許左IR輸送補助氣缸下降
      ANI     L4700  ; 左側合流補助昇降下降定點
      OUT     B1144  ; 左側合流補助昇降下降
6297  LD      B1144  ; 左側合流補助昇降下降
      OUT     B264  ; 左IR輸送出框補助氣缸C13下降SV
6299  LD      B1144  ; 左側合流補助昇降下降
      AND     SM412  ; 1.0 Sec Clock
      OR      L4700  ; 左側合流補助昇降下降定點
      OUT     M344  ; 左IR輸送出框氣缸伸出燈
6303  LD      L4027  ; 出料機構允許運轉
      ANDPI   M4132  ; 左側合流補助昇降異常
      OUT     L145  ; 允許左IR輸送出框氣缸縮回
6307  LD      M145  ; 左IR輸送出框氣缸縮回SW
      ANI     L4315  ; 出料合流機構回原點
      LDI     L4891  ; 出料分流左側取框原點
      AND     L4315  ; 出料合流機構回原點
      AND     L4740  ; 出料合流左側伸出伸出定點
      AND     L4742  ; 出料合流左側昇降上定點
      AND     L4706  ; 左IR輸送出框定點有框
      ORB
      AND     L3653  ; 出料手動允許信號
      AND     L145  ; 允許左IR輸送出框氣缸縮回
      OUT     T145 D106  ; 手動左IR輸送出框氣缸縮回延遲
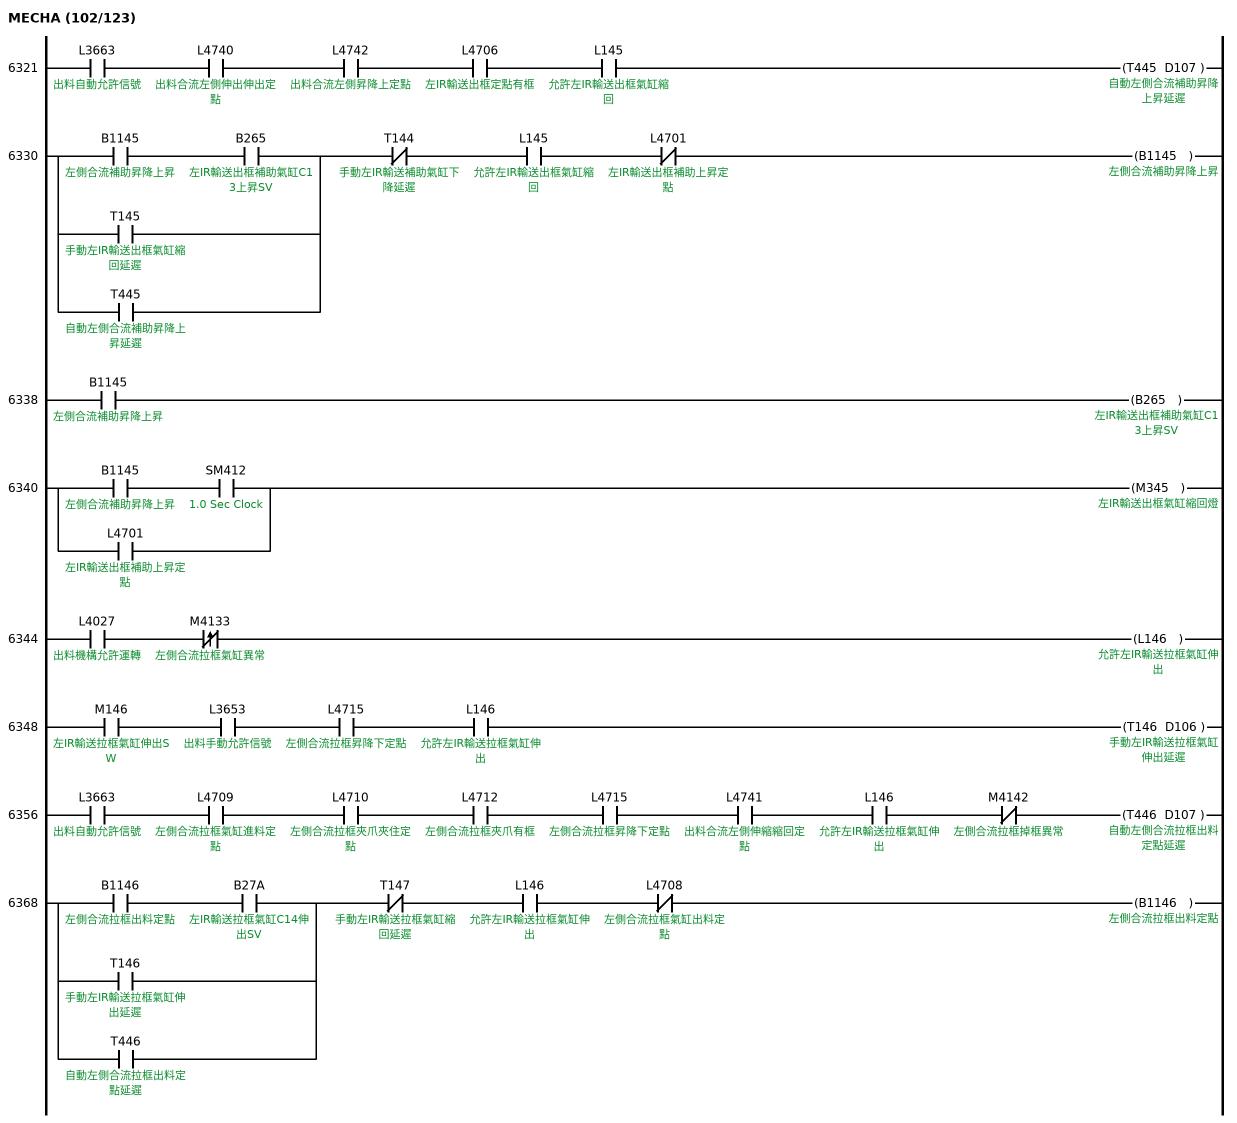
6321  LD      L3663  ; 出料自動允許信號
      AND     L4740  ; 出料合流左側伸出伸出定點
      AND     L4742  ; 出料合流左側昇降上定點
      AND     L4706  ; 左IR輸送出框定點有框
      AND     L145  ; 允許左IR輸送出框氣缸縮回
      OUT     T445 D107  ; 自動左側合流補助昇降上昇延遲
6330  LD      B1145  ; 左側合流補助昇降上昇
      AND     B265  ; 左IR輸送出框補助氣缸C13上昇SV
      OR      T145  ; 手動左IR輸送出框氣缸縮回延遲
      OR      T445  ; 自動左側合流補助昇降上昇延遲
      ANI     T144  ; 手動左IR輸送補助氣缸下降延遲
      AND     L145  ; 允許左IR輸送出框氣缸縮回
      ANI     L4701  ; 左IR輸送出框補助上昇定點
      OUT     B1145  ; 左側合流補助昇降上昇
6338  LD      B1145  ; 左側合流補助昇降上昇
      OUT     B265  ; 左IR輸送出框補助氣缸C13上昇SV
6340  LD      B1145  ; 左側合流補助昇降上昇
      AND     SM412  ; 1.0 Sec Clock
      OR      L4701  ; 左IR輸送出框補助上昇定點
      OUT     M345  ; 左IR輸送出框氣缸縮回燈
6344  LD      L4027  ; 出料機構允許運轉
      ANDPI   M4133  ; 左側合流拉框氣缸異常
      OUT     L146  ; 允許左IR輸送拉框氣缸伸出
6348  LD      M146  ; 左IR輸送拉框氣缸伸出SW
      AND     L3653  ; 出料手動允許信號
      AND     L4715  ; 左側合流拉框昇降下定點
      AND     L146  ; 允許左IR輸送拉框氣缸伸出
      OUT     T146 D106  ; 手動左IR輸送拉框氣缸伸出延遲
6356  LD      L3663  ; 出料自動允許信號
      AND     L4709  ; 左側合流拉框氣缸進料定點
      AND     L4710  ; 左側合流拉框夾爪夾住定點
      AND     L4712  ; 左側合流拉框夾爪有框
      AND     L4715  ; 左側合流拉框昇降下定點
      AND     L4741  ; 出料合流左側伸縮縮回定點
      AND     L146  ; 允許左IR輸送拉框氣缸伸出
      ANI     M4142  ; 左側合流拉框掉框異常
      OUT     T446 D107  ; 自動左側合流拉框出料定點延遲
6368  LD      B1146  ; 左側合流拉框出料定點
      AND     B27A  ; 左IR輸送拉框氣缸C14伸出SV
      OR      T146  ; 手動左IR輸送拉框氣缸伸出延遲
      OR      T446  ; 自動左側合流拉框出料定點延遲
      ANI     T147  ; 手動左IR輸送拉框氣缸縮回延遲
      AND     L146  ; 允許左IR輸送拉框氣缸伸出
      ANI     L4708  ; 左側合流拉框氣缸出料定點
      OUT     B1146  ; 左側合流拉框出料定點
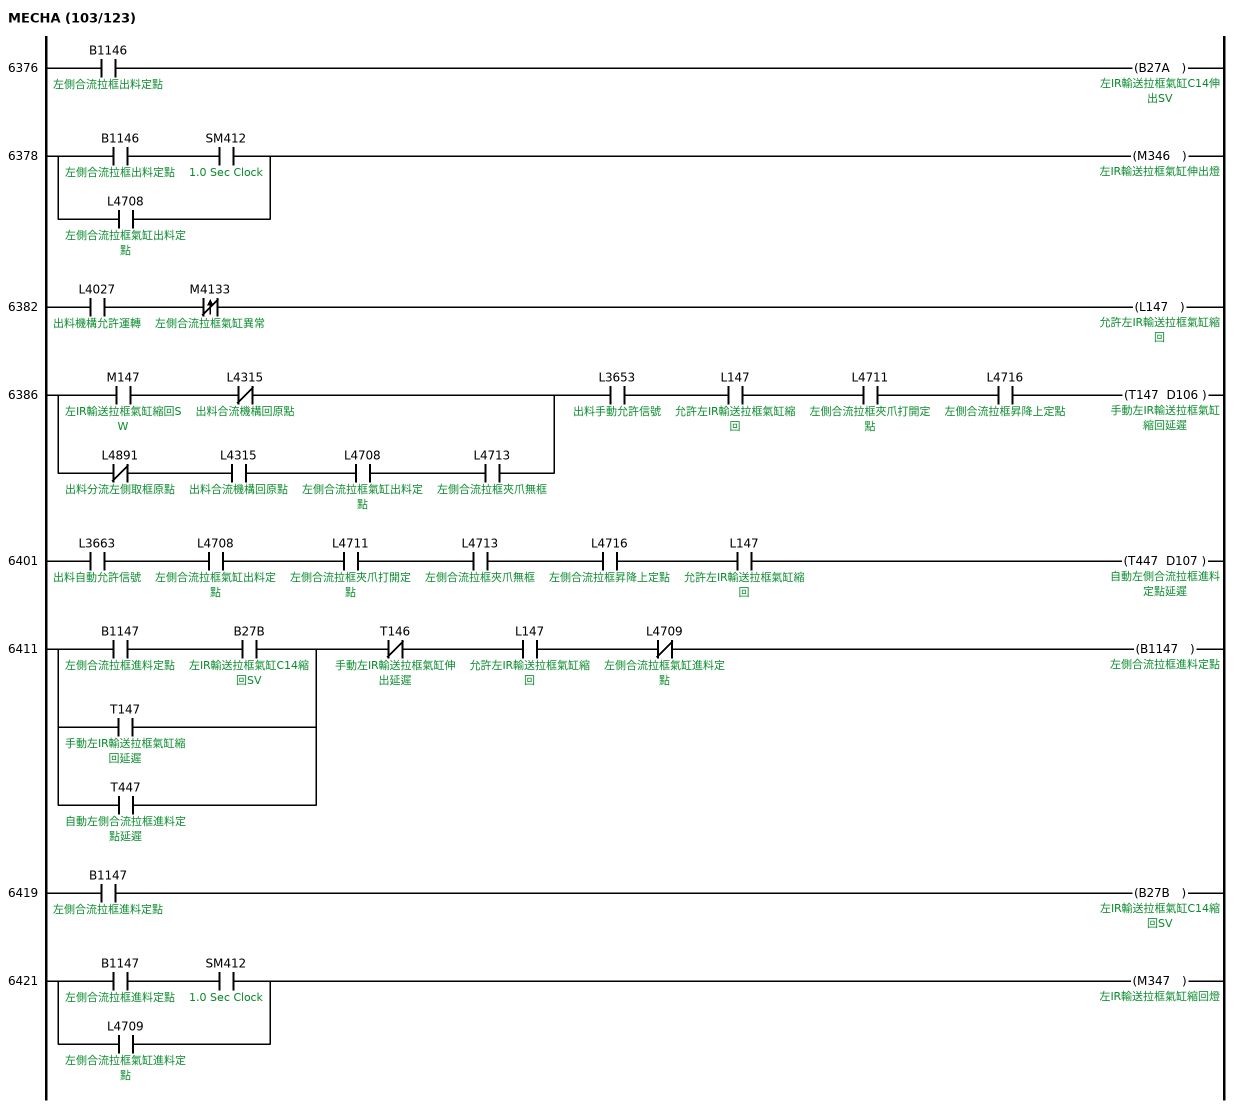
6376  LD      B1146  ; 左側合流拉框出料定點
      OUT     B27A  ; 左IR輸送拉框氣缸C14伸出SV
6378  LD      B1146  ; 左側合流拉框出料定點
      AND     SM412  ; 1.0 Sec Clock
      OR      L4708  ; 左側合流拉框氣缸出料定點
      OUT     M346  ; 左IR輸送拉框氣缸伸出燈
6382  LD      L4027  ; 出料機構允許運轉
      ANDPI   M4133  ; 左側合流拉框氣缸異常
      OUT     L147  ; 允許左IR輸送拉框氣缸縮回
6386  LD      M147  ; 左IR輸送拉框氣缸縮回SW
      ANI     L4315  ; 出料合流機構回原點
      LDI     L4891  ; 出料分流左側取框原點
      AND     L4315  ; 出料合流機構回原點
      AND     L4708  ; 左側合流拉框氣缸出料定點
      AND     L4713  ; 左側合流拉框夾爪無框
      ORB
      AND     L3653  ; 出料手動允許信號
      AND     L147  ; 允許左IR輸送拉框氣缸縮回
      AND     L4711  ; 左側合流拉框夾爪打開定點
      AND     L4716  ; 左側合流拉框昇降上定點
      OUT     T147 D106  ; 手動左IR輸送拉框氣缸縮回延遲
6401  LD      L3663  ; 出料自動允許信號
      AND     L4708  ; 左側合流拉框氣缸出料定點
      AND     L4711  ; 左側合流拉框夾爪打開定點
      AND     L4713  ; 左側合流拉框夾爪無框
      AND     L4716  ; 左側合流拉框昇降上定點
      AND     L147  ; 允許左IR輸送拉框氣缸縮回
      OUT     T447 D107  ; 自動左側合流拉框進料定點延遲
6411  LD      B1147  ; 左側合流拉框進料定點
      AND     B27B  ; 左IR輸送拉框氣缸C14縮回SV
      OR      T147  ; 手動左IR輸送拉框氣缸縮回延遲
      OR      T447  ; 自動左側合流拉框進料定點延遲
      ANI     T146  ; 手動左IR輸送拉框氣缸伸出延遲
      AND     L147  ; 允許左IR輸送拉框氣缸縮回
      ANI     L4709  ; 左側合流拉框氣缸進料定點
      OUT     B1147  ; 左側合流拉框進料定點
6419  LD      B1147  ; 左側合流拉框進料定點
      OUT     B27B  ; 左IR輸送拉框氣缸C14縮回SV
6421  LD      B1147  ; 左側合流拉框進料定點
      AND     SM412  ; 1.0 Sec Clock
      OR      L4709  ; 左側合流拉框氣缸進料定點
      OUT     M347  ; 左IR輸送拉框氣缸縮回燈
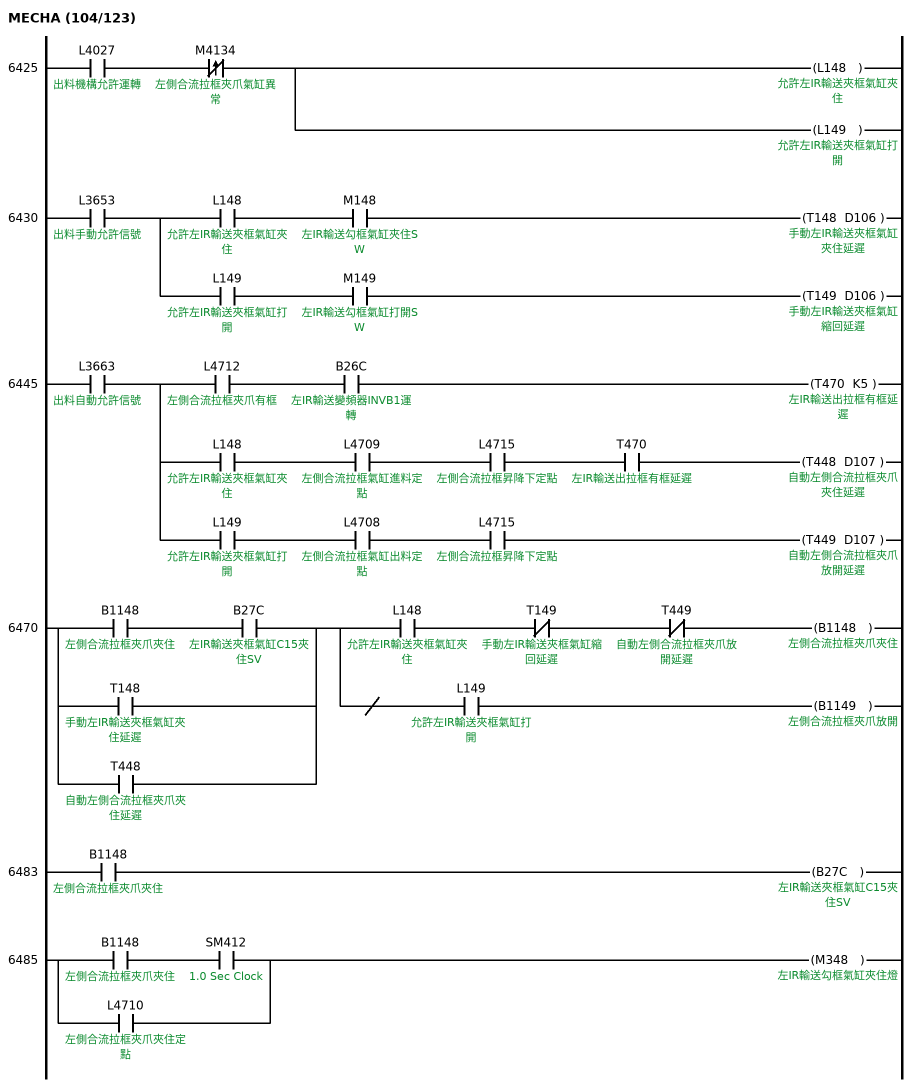
6425  LD      L4027  ; 出料機構允許運轉
      ANDPI   M4134  ; 左側合流拉框夾爪氣缸異常
      OUT     L148  ; 允許左IR輸送夾框氣缸夾住
      OUT     L149  ; 允許左IR輸送夾框氣缸打開
6430  LD      L3653  ; 出料手動允許信號
      MPS
      AND     L148  ; 允許左IR輸送夾框氣缸夾住
      AND     M148  ; 左IR輸送勾框氣缸夾住SW
      OUT     T148 D106  ; 手動左IR輸送夾框氣缸夾住延遲
      MPP
      AND     L149  ; 允許左IR輸送夾框氣缸打開
      AND     M149  ; 左IR輸送勾框氣缸打開SW
      OUT     T149 D106  ; 手動左IR輸送夾框氣缸縮回延遲
6445  LD      L3663  ; 出料自動允許信號
      MPS
      AND     L4712  ; 左側合流拉框夾爪有框
      AND     B26C  ; 左IR輸送變頻器INVB1運轉
      OUT     T470 K5  ; 左IR輸送出拉框有框延遲
      MRD
      AND     L148  ; 允許左IR輸送夾框氣缸夾住
      AND     L4709  ; 左側合流拉框氣缸進料定點
      AND     L4715  ; 左側合流拉框昇降下定點
      AND     T470  ; 左IR輸送出拉框有框延遲
      OUT     T448 D107  ; 自動左側合流拉框夾爪夾住延遲
      MPP
      AND     L149  ; 允許左IR輸送夾框氣缸打開
      AND     L4708  ; 左側合流拉框氣缸出料定點
      AND     L4715  ; 左側合流拉框昇降下定點
      OUT     T449 D107  ; 自動左側合流拉框夾爪放開延遲
6470  LD      B1148  ; 左側合流拉框夾爪夾住
      AND     B27C  ; 左IR輸送夾框氣缸C15夾住SV
      OR      T148  ; 手動左IR輸送夾框氣缸夾住延遲
      OR      T448  ; 自動左側合流拉框夾爪夾住延遲
      MPS
      AND     L148  ; 允許左IR輸送夾框氣缸夾住
      ANI     T149  ; 手動左IR輸送夾框氣缸縮回延遲
      ANI     T449  ; 自動左側合流拉框夾爪放開延遲
      OUT     B1148  ; 左側合流拉框夾爪夾住
      MPP
      INV
      AND     L149  ; 允許左IR輸送夾框氣缸打開
      OUT     B1149  ; 左側合流拉框夾爪放開
6483  LD      B1148  ; 左側合流拉框夾爪夾住
      OUT     B27C  ; 左IR輸送夾框氣缸C15夾住SV
6485  LD      B1148  ; 左側合流拉框夾爪夾住
      AND     SM412  ; 1.0 Sec Clock
      OR      L4710  ; 左側合流拉框夾爪夾住定點
      OUT     M348  ; 左IR輸送勾框氣缸夾住燈
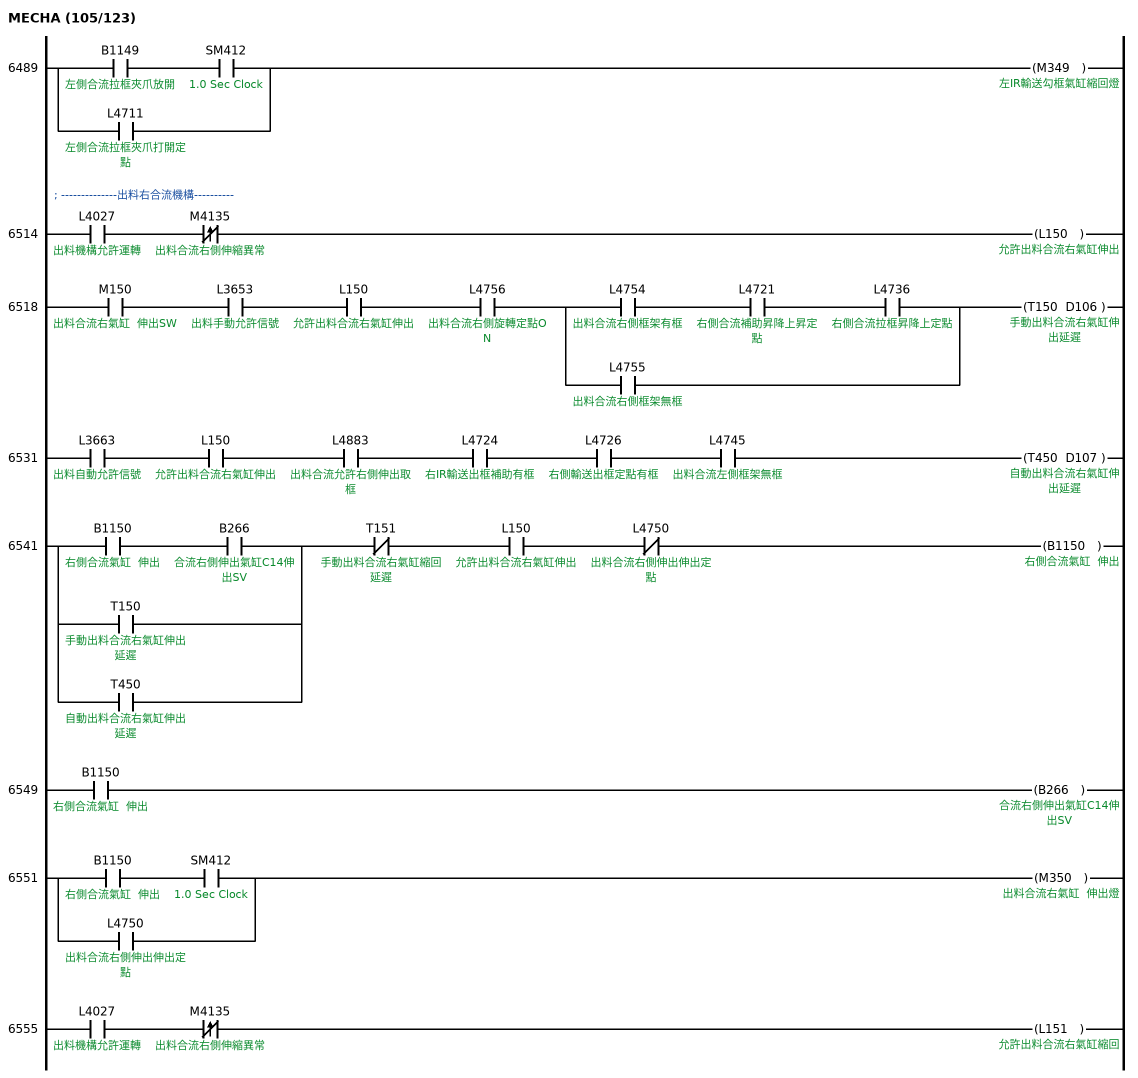
6489  LD      B1149  ; 左側合流拉框夾爪放開
      AND     SM412  ; 1.0 Sec Clock
      OR      L4711  ; 左側合流拉框夾爪打開定點
      OUT     M349  ; 左IR輸送勾框氣缸縮回燈
; --------------出料右合流機構----------
6514  LD      L4027  ; 出料機構允許運轉
      ANDPI   M4135  ; 出料合流右側伸縮異常
      OUT     L150  ; 允許出料合流右氣缸伸出
6518  LD      M150  ; 出料合流右氣缸  伸出SW
      AND     L3653  ; 出料手動允許信號
      AND     L150  ; 允許出料合流右氣缸伸出
      AND     L4756  ; 出料合流右側旋轉定點ON
      LD      L4754  ; 出料合流右側框架有框
      AND     L4721  ; 右側合流補助昇降上昇定點
      AND     L4736  ; 右側合流拉框昇降上定點
      OR      L4755  ; 出料合流右側框架無框
      ANB
      OUT     T150 D106  ; 手動出料合流右氣缸伸出延遲
6531  LD      L3663  ; 出料自動允許信號
      AND     L150  ; 允許出料合流右氣缸伸出
      AND     L4883  ; 出料合流允許右側伸出取框
      AND     L4724  ; 右IR輸送出框補助有框
      AND     L4726  ; 右側輸送出框定點有框
      AND     L4745  ; 出料合流左側框架無框
      OUT     T450 D107  ; 自動出料合流右氣缸伸出延遲
6541  LD      B1150  ; 右側合流氣缸  伸出
      AND     B266  ; 合流右側伸出氣缸C14伸出SV
      OR      T150  ; 手動出料合流右氣缸伸出延遲
      OR      T450  ; 自動出料合流右氣缸伸出延遲
      ANI     T151  ; 手動出料合流右氣缸縮回延遲
      AND     L150  ; 允許出料合流右氣缸伸出
      ANI     L4750  ; 出料合流右側伸出伸出定點
      OUT     B1150  ; 右側合流氣缸  伸出
6549  LD      B1150  ; 右側合流氣缸  伸出
      OUT     B266  ; 合流右側伸出氣缸C14伸出SV
6551  LD      B1150  ; 右側合流氣缸  伸出
      AND     SM412  ; 1.0 Sec Clock
      OR      L4750  ; 出料合流右側伸出伸出定點
      OUT     M350  ; 出料合流右氣缸  伸出燈
6555  LD      L4027  ; 出料機構允許運轉
      ANDPI   M4135  ; 出料合流右側伸縮異常
      OUT     L151  ; 允許出料合流右氣缸縮回
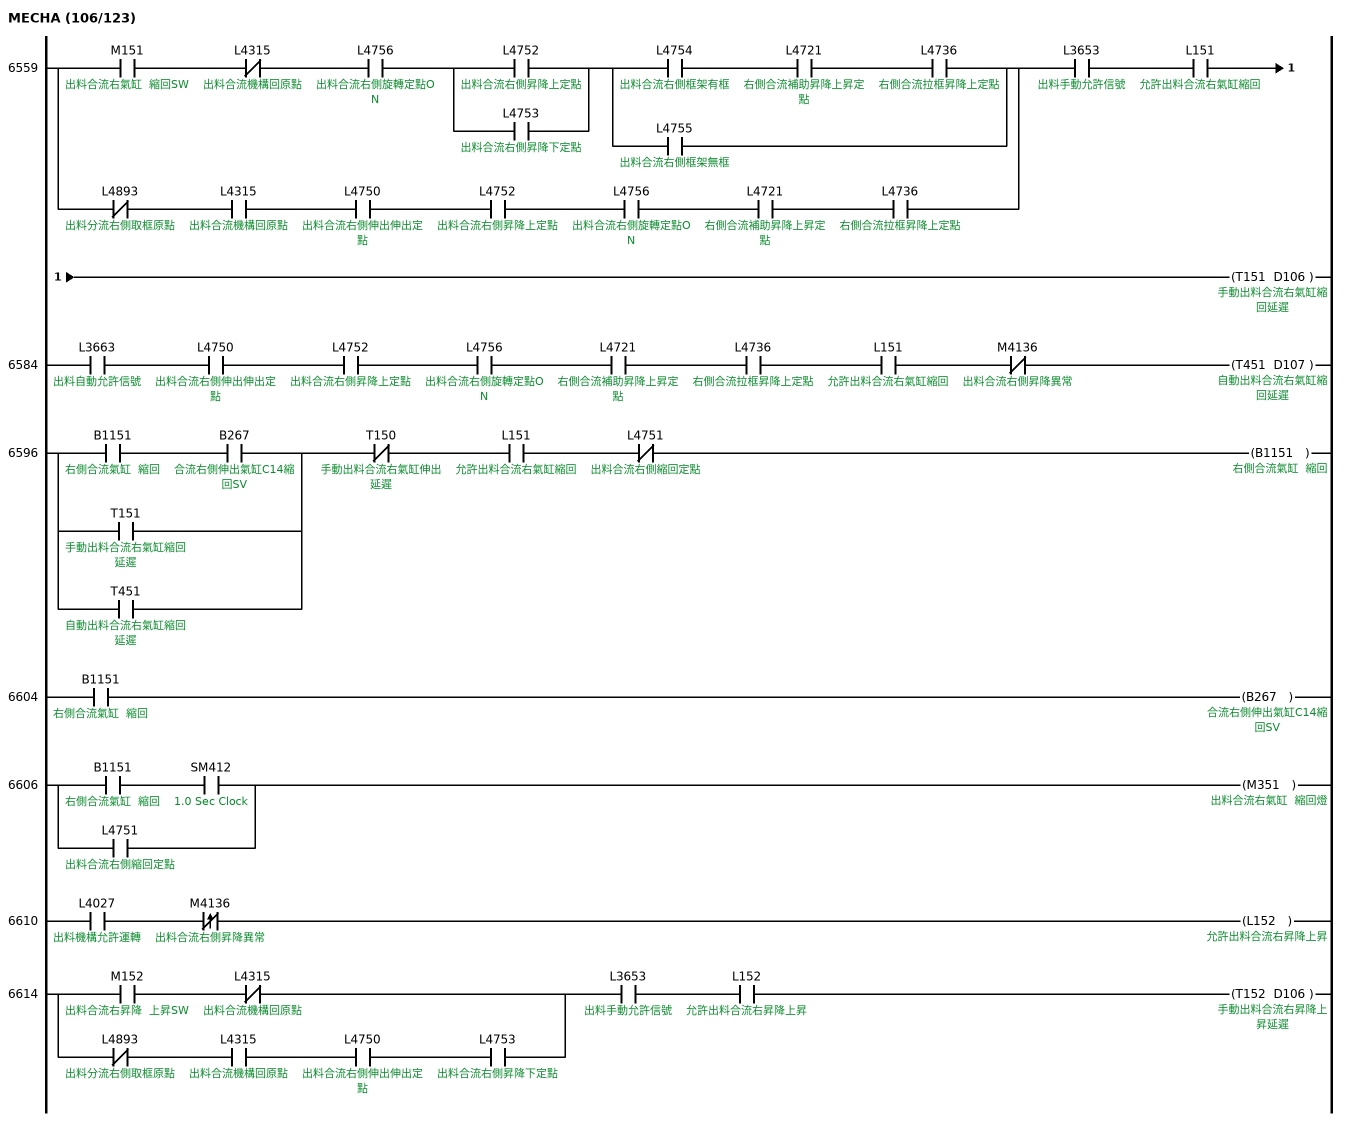
6559  LD      M151  ; 出料合流右氣缸  縮回SW
      ANI     L4315  ; 出料合流機構回原點
      AND     L4756  ; 出料合流右側旋轉定點ON
      LD      L4752  ; 出料合流右側昇降上定點
      OR      L4753  ; 出料合流右側昇降下定點
      ANB
      LD      L4754  ; 出料合流右側框架有框
      AND     L4721  ; 右側合流補助昇降上昇定點
      AND     L4736  ; 右側合流拉框昇降上定點
      OR      L4755  ; 出料合流右側框架無框
      ANB
      LDI     L4893  ; 出料分流右側取框原點
      AND     L4315  ; 出料合流機構回原點
      AND     L4750  ; 出料合流右側伸出伸出定點
      AND     L4752  ; 出料合流右側昇降上定點
      AND     L4756  ; 出料合流右側旋轉定點ON
      AND     L4721  ; 右側合流補助昇降上昇定點
      AND     L4736  ; 右側合流拉框昇降上定點
      ORB
      AND     L3653  ; 出料手動允許信號
      AND     L151  ; 允許出料合流右氣缸縮回
      OUT     T151 D106  ; 手動出料合流右氣缸縮回延遲
6584  LD      L3663  ; 出料自動允許信號
      AND     L4750  ; 出料合流右側伸出伸出定點
      AND     L4752  ; 出料合流右側昇降上定點
      AND     L4756  ; 出料合流右側旋轉定點ON
      AND     L4721  ; 右側合流補助昇降上昇定點
      AND     L4736  ; 右側合流拉框昇降上定點
      AND     L151  ; 允許出料合流右氣缸縮回
      ANI     M4136  ; 出料合流右側昇降異常
      OUT     T451 D107  ; 自動出料合流右氣缸縮回延遲
6596  LD      B1151  ; 右側合流氣缸  縮回
      AND     B267  ; 合流右側伸出氣缸C14縮回SV
      OR      T151  ; 手動出料合流右氣缸縮回延遲
      OR      T451  ; 自動出料合流右氣缸縮回延遲
      ANI     T150  ; 手動出料合流右氣缸伸出延遲
      AND     L151  ; 允許出料合流右氣缸縮回
      ANI     L4751  ; 出料合流右側縮回定點
      OUT     B1151  ; 右側合流氣缸  縮回
6604  LD      B1151  ; 右側合流氣缸  縮回
      OUT     B267  ; 合流右側伸出氣缸C14縮回SV
6606  LD      B1151  ; 右側合流氣缸  縮回
      AND     SM412  ; 1.0 Sec Clock
      OR      L4751  ; 出料合流右側縮回定點
      OUT     M351  ; 出料合流右氣缸  縮回燈
6610  LD      L4027  ; 出料機構允許運轉
      ANDPI   M4136  ; 出料合流右側昇降異常
      OUT     L152  ; 允許出料合流右昇降上昇
6614  LD      M152  ; 出料合流右昇降  上昇SW
      ANI     L4315  ; 出料合流機構回原點
      LDI     L4893  ; 出料分流右側取框原點
      AND     L4315  ; 出料合流機構回原點
      AND     L4750  ; 出料合流右側伸出伸出定點
      AND     L4753  ; 出料合流右側昇降下定點
      ORB
      AND     L3653  ; 出料手動允許信號
      AND     L152  ; 允許出料合流右昇降上昇
      OUT     T152 D106  ; 手動出料合流右昇降上昇延遲
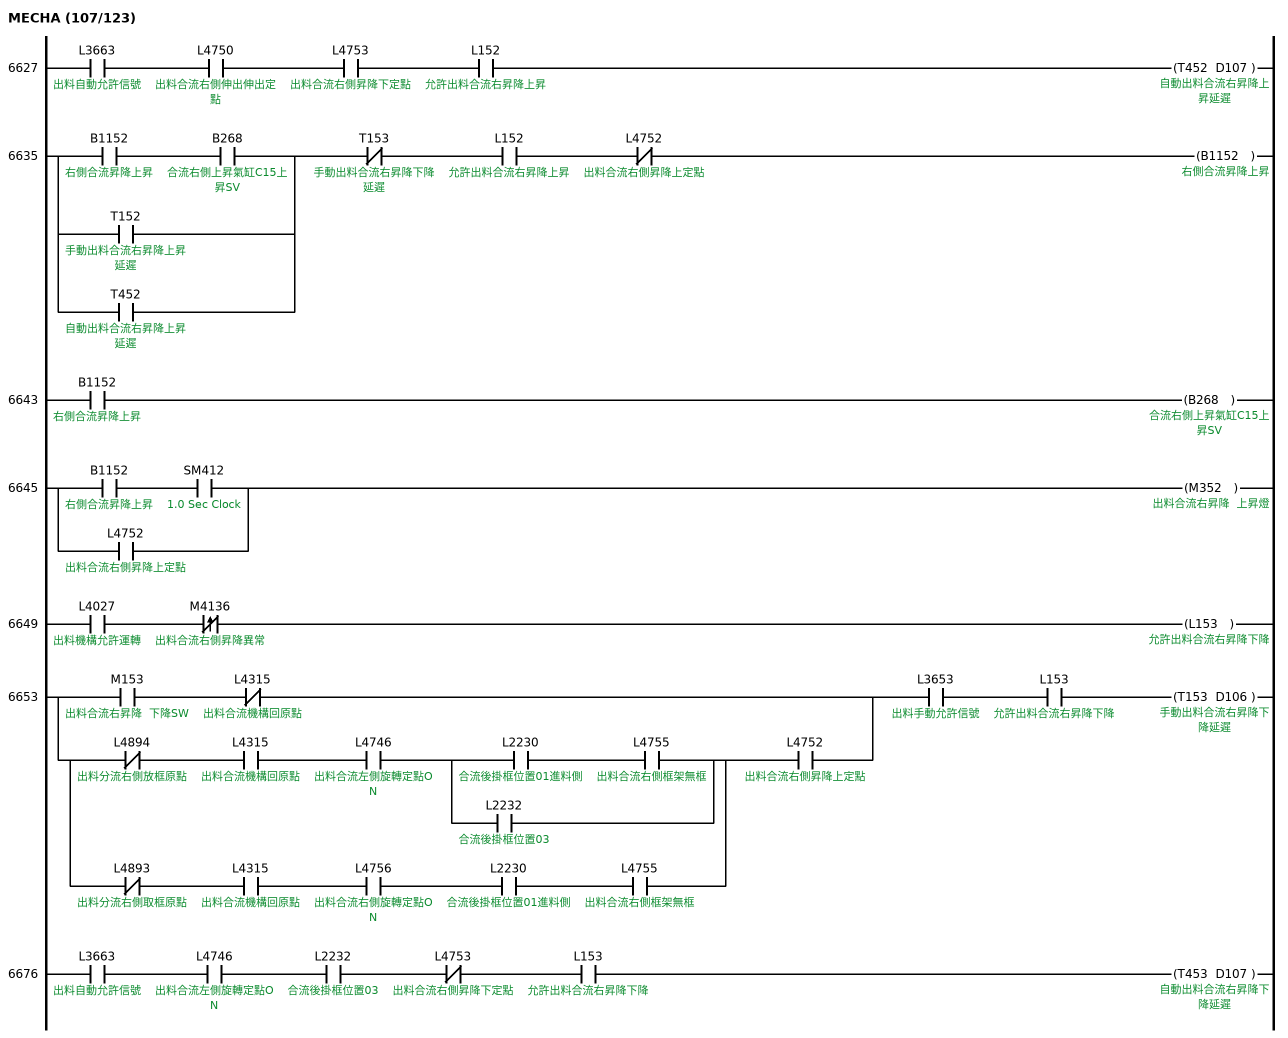
6627  LD      L3663  ; 出料自動允許信號
      AND     L4750  ; 出料合流右側伸出伸出定點
      AND     L4753  ; 出料合流右側昇降下定點
      AND     L152  ; 允許出料合流右昇降上昇
      OUT     T452 D107  ; 自動出料合流右昇降上昇延遲
6635  LD      B1152  ; 右側合流昇降上昇
      AND     B268  ; 合流右側上昇氣缸C15上昇SV
      OR      T152  ; 手動出料合流右昇降上昇延遲
      OR      T452  ; 自動出料合流右昇降上昇延遲
      ANI     T153  ; 手動出料合流右昇降下降延遲
      AND     L152  ; 允許出料合流右昇降上昇
      ANI     L4752  ; 出料合流右側昇降上定點
      OUT     B1152  ; 右側合流昇降上昇
6643  LD      B1152  ; 右側合流昇降上昇
      OUT     B268  ; 合流右側上昇氣缸C15上昇SV
6645  LD      B1152  ; 右側合流昇降上昇
      AND     SM412  ; 1.0 Sec Clock
      OR      L4752  ; 出料合流右側昇降上定點
      OUT     M352  ; 出料合流右昇降  上昇燈
6649  LD      L4027  ; 出料機構允許運轉
      ANDPI   M4136  ; 出料合流右側昇降異常
      OUT     L153  ; 允許出料合流右昇降下降
6653  LD      M153  ; 出料合流右昇降  下降SW
      ANI     L4315  ; 出料合流機構回原點
      LDI     L4894  ; 出料分流右側放框原點
      AND     L4315  ; 出料合流機構回原點
      AND     L4746  ; 出料合流左側旋轉定點ON
      LD      L2230  ; 合流後掛框位置01進料側
      AND     L4755  ; 出料合流右側框架無框
      OR      L2232  ; 合流後掛框位置03
      ANB
      LDI     L4893  ; 出料分流右側取框原點
      AND     L4315  ; 出料合流機構回原點
      AND     L4756  ; 出料合流右側旋轉定點ON
      AND     L2230  ; 合流後掛框位置01進料側
      AND     L4755  ; 出料合流右側框架無框
      ORB
      AND     L4752  ; 出料合流右側昇降上定點
      ORB
      AND     L3653  ; 出料手動允許信號
      AND     L153  ; 允許出料合流右昇降下降
      OUT     T153 D106  ; 手動出料合流右昇降下降延遲
6676  LD      L3663  ; 出料自動允許信號
      AND     L4746  ; 出料合流左側旋轉定點ON
      AND     L2232  ; 合流後掛框位置03
      ANI     L4753  ; 出料合流右側昇降下定點
      AND     L153  ; 允許出料合流右昇降下降
      OUT     T453 D107  ; 自動出料合流右昇降下降延遲
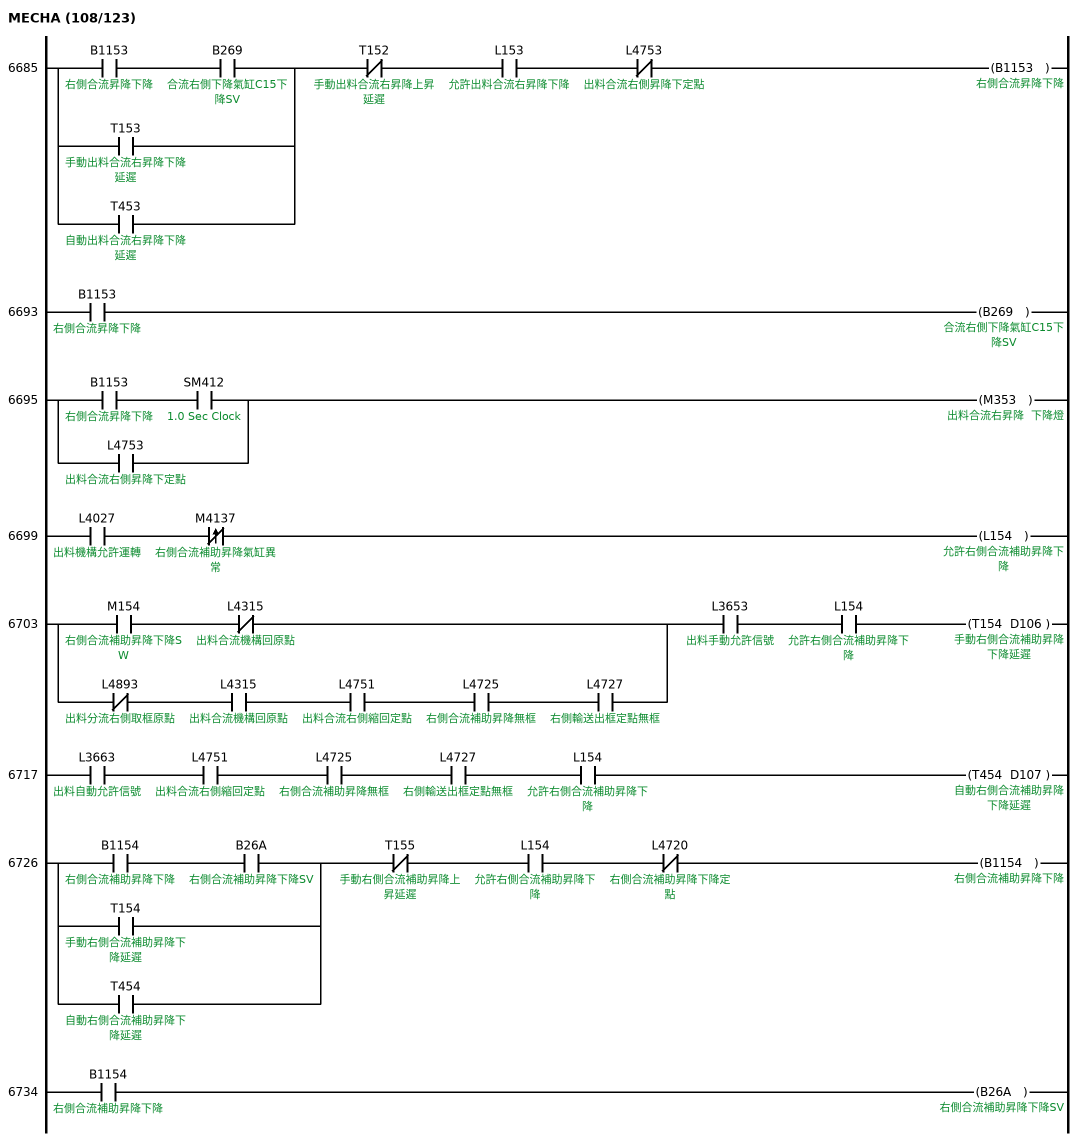
6685  LD      B1153  ; 右側合流昇降下降
      AND     B269  ; 合流右側下降氣缸C15下降SV
      OR      T153  ; 手動出料合流右昇降下降延遲
      OR      T453  ; 自動出料合流右昇降下降延遲
      ANI     T152  ; 手動出料合流右昇降上昇延遲
      AND     L153  ; 允許出料合流右昇降下降
      ANI     L4753  ; 出料合流右側昇降下定點
      OUT     B1153  ; 右側合流昇降下降
6693  LD      B1153  ; 右側合流昇降下降
      OUT     B269  ; 合流右側下降氣缸C15下降SV
6695  LD      B1153  ; 右側合流昇降下降
      AND     SM412  ; 1.0 Sec Clock
      OR      L4753  ; 出料合流右側昇降下定點
      OUT     M353  ; 出料合流右昇降  下降燈
6699  LD      L4027  ; 出料機構允許運轉
      ANDPI   M4137  ; 右側合流補助昇降氣缸異常
      OUT     L154  ; 允許右側合流補助昇降下降
6703  LD      M154  ; 右側合流補助昇降下降SW
      ANI     L4315  ; 出料合流機構回原點
      LDI     L4893  ; 出料分流右側取框原點
      AND     L4315  ; 出料合流機構回原點
      AND     L4751  ; 出料合流右側縮回定點
      AND     L4725  ; 右側合流補助昇降無框
      AND     L4727  ; 右側輸送出框定點無框
      ORB
      AND     L3653  ; 出料手動允許信號
      AND     L154  ; 允許右側合流補助昇降下降
      OUT     T154 D106  ; 手動右側合流補助昇降下降延遲
6717  LD      L3663  ; 出料自動允許信號
      AND     L4751  ; 出料合流右側縮回定點
      AND     L4725  ; 右側合流補助昇降無框
      AND     L4727  ; 右側輸送出框定點無框
      AND     L154  ; 允許右側合流補助昇降下降
      OUT     T454 D107  ; 自動右側合流補助昇降下降延遲
6726  LD      B1154  ; 右側合流補助昇降下降
      AND     B26A  ; 右側合流補助昇降下降SV
      OR      T154  ; 手動右側合流補助昇降下降延遲
      OR      T454  ; 自動右側合流補助昇降下降延遲
      ANI     T155  ; 手動右側合流補助昇降上昇延遲
      AND     L154  ; 允許右側合流補助昇降下降
      ANI     L4720  ; 右側合流補助昇降下降定點
      OUT     B1154  ; 右側合流補助昇降下降
6734  LD      B1154  ; 右側合流補助昇降下降
      OUT     B26A  ; 右側合流補助昇降下降SV
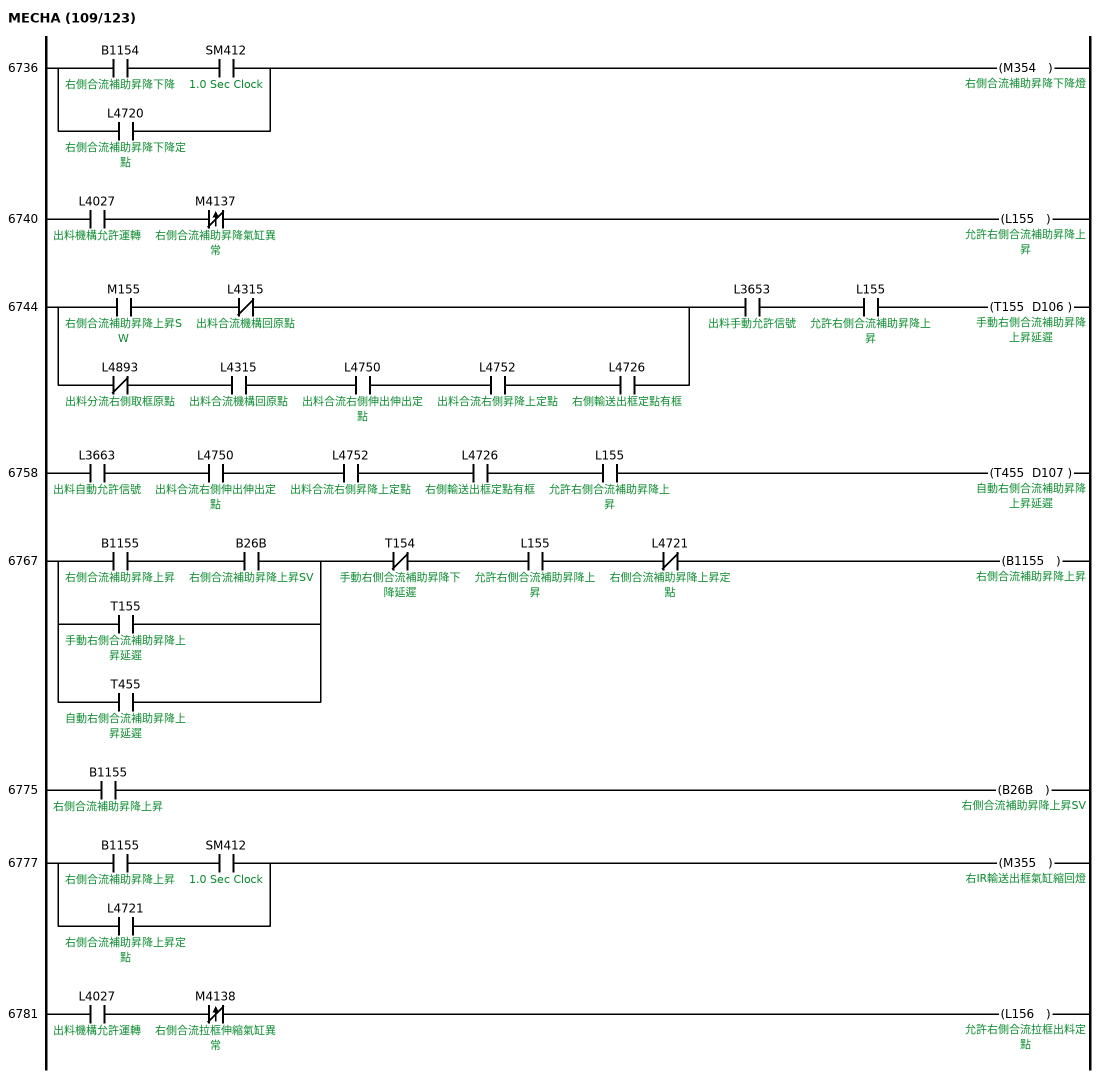
6736  LD      B1154  ; 右側合流補助昇降下降
      AND     SM412  ; 1.0 Sec Clock
      OR      L4720  ; 右側合流補助昇降下降定點
      OUT     M354  ; 右側合流補助昇降下降燈
6740  LD      L4027  ; 出料機構允許運轉
      ANDPI   M4137  ; 右側合流補助昇降氣缸異常
      OUT     L155  ; 允許右側合流補助昇降上昇
6744  LD      M155  ; 右側合流補助昇降上昇SW
      ANI     L4315  ; 出料合流機構回原點
      LDI     L4893  ; 出料分流右側取框原點
      AND     L4315  ; 出料合流機構回原點
      AND     L4750  ; 出料合流右側伸出伸出定點
      AND     L4752  ; 出料合流右側昇降上定點
      AND     L4726  ; 右側輸送出框定點有框
      ORB
      AND     L3653  ; 出料手動允許信號
      AND     L155  ; 允許右側合流補助昇降上昇
      OUT     T155 D106  ; 手動右側合流補助昇降上昇延遲
6758  LD      L3663  ; 出料自動允許信號
      AND     L4750  ; 出料合流右側伸出伸出定點
      AND     L4752  ; 出料合流右側昇降上定點
      AND     L4726  ; 右側輸送出框定點有框
      AND     L155  ; 允許右側合流補助昇降上昇
      OUT     T455 D107  ; 自動右側合流補助昇降上昇延遲
6767  LD      B1155  ; 右側合流補助昇降上昇
      AND     B26B  ; 右側合流補助昇降上昇SV
      OR      T155  ; 手動右側合流補助昇降上昇延遲
      OR      T455  ; 自動右側合流補助昇降上昇延遲
      ANI     T154  ; 手動右側合流補助昇降下降延遲
      AND     L155  ; 允許右側合流補助昇降上昇
      ANI     L4721  ; 右側合流補助昇降上昇定點
      OUT     B1155  ; 右側合流補助昇降上昇
6775  LD      B1155  ; 右側合流補助昇降上昇
      OUT     B26B  ; 右側合流補助昇降上昇SV
6777  LD      B1155  ; 右側合流補助昇降上昇
      AND     SM412  ; 1.0 Sec Clock
      OR      L4721  ; 右側合流補助昇降上昇定點
      OUT     M355  ; 右IR輸送出框氣缸縮回燈
6781  LD      L4027  ; 出料機構允許運轉
      ANDPI   M4138  ; 右側合流拉框伸縮氣缸異常
      OUT     L156  ; 允許右側合流拉框出料定點
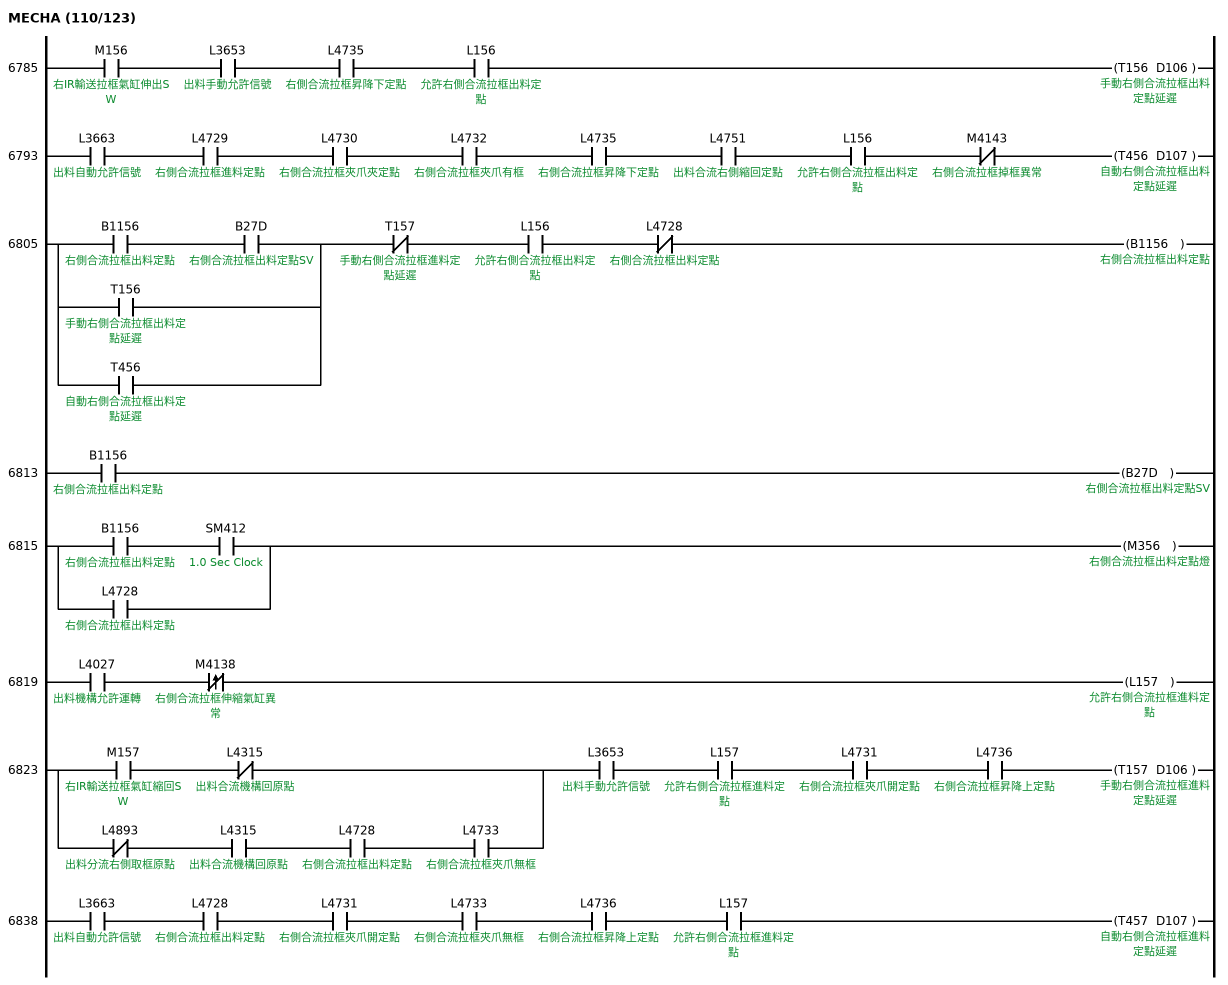
6785  LD      M156  ; 右IR輸送拉框氣缸伸出SW
      AND     L3653  ; 出料手動允許信號
      AND     L4735  ; 右側合流拉框昇降下定點
      AND     L156  ; 允許右側合流拉框出料定點
      OUT     T156 D106  ; 手動右側合流拉框出料定點延遲
6793  LD      L3663  ; 出料自動允許信號
      AND     L4729  ; 右側合流拉框進料定點
      AND     L4730  ; 右側合流拉框夾爪夾定點
      AND     L4732  ; 右側合流拉框夾爪有框
      AND     L4735  ; 右側合流拉框昇降下定點
      AND     L4751  ; 出料合流右側縮回定點
      AND     L156  ; 允許右側合流拉框出料定點
      ANI     M4143  ; 右側合流拉框掉框異常
      OUT     T456 D107  ; 自動右側合流拉框出料定點延遲
6805  LD      B1156  ; 右側合流拉框出料定點
      AND     B27D  ; 右側合流拉框出料定點SV
      OR      T156  ; 手動右側合流拉框出料定點延遲
      OR      T456  ; 自動右側合流拉框出料定點延遲
      ANI     T157  ; 手動右側合流拉框進料定點延遲
      AND     L156  ; 允許右側合流拉框出料定點
      ANI     L4728  ; 右側合流拉框出料定點
      OUT     B1156  ; 右側合流拉框出料定點
6813  LD      B1156  ; 右側合流拉框出料定點
      OUT     B27D  ; 右側合流拉框出料定點SV
6815  LD      B1156  ; 右側合流拉框出料定點
      AND     SM412  ; 1.0 Sec Clock
      OR      L4728  ; 右側合流拉框出料定點
      OUT     M356  ; 右側合流拉框出料定點燈
6819  LD      L4027  ; 出料機構允許運轉
      ANDPI   M4138  ; 右側合流拉框伸縮氣缸異常
      OUT     L157  ; 允許右側合流拉框進料定點
6823  LD      M157  ; 右IR輸送拉框氣缸縮回SW
      ANI     L4315  ; 出料合流機構回原點
      LDI     L4893  ; 出料分流右側取框原點
      AND     L4315  ; 出料合流機構回原點
      AND     L4728  ; 右側合流拉框出料定點
      AND     L4733  ; 右側合流拉框夾爪無框
      ORB
      AND     L3653  ; 出料手動允許信號
      AND     L157  ; 允許右側合流拉框進料定點
      AND     L4731  ; 右側合流拉框夾爪開定點
      AND     L4736  ; 右側合流拉框昇降上定點
      OUT     T157 D106  ; 手動右側合流拉框進料定點延遲
6838  LD      L3663  ; 出料自動允許信號
      AND     L4728  ; 右側合流拉框出料定點
      AND     L4731  ; 右側合流拉框夾爪開定點
      AND     L4733  ; 右側合流拉框夾爪無框
      AND     L4736  ; 右側合流拉框昇降上定點
      AND     L157  ; 允許右側合流拉框進料定點
      OUT     T457 D107  ; 自動右側合流拉框進料定點延遲
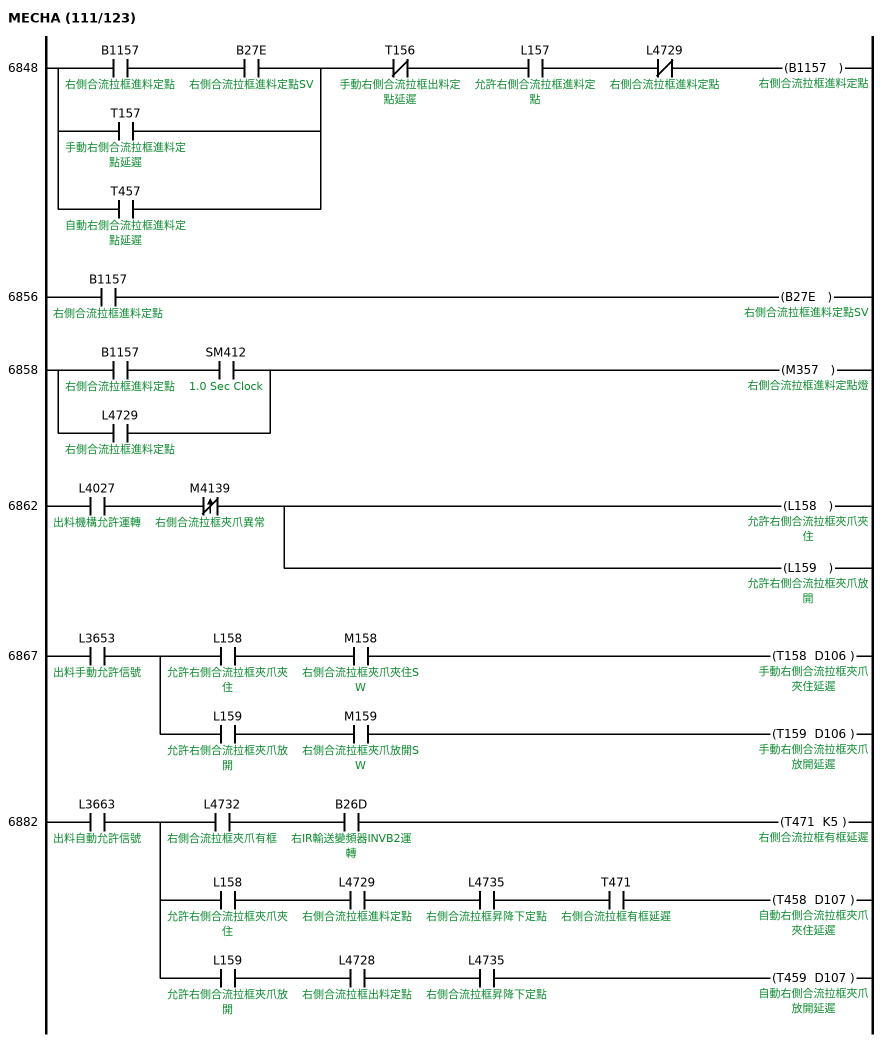
6848  LD      B1157  ; 右側合流拉框進料定點
      AND     B27E  ; 右側合流拉框進料定點SV
      OR      T157  ; 手動右側合流拉框進料定點延遲
      OR      T457  ; 自動右側合流拉框進料定點延遲
      ANI     T156  ; 手動右側合流拉框出料定點延遲
      AND     L157  ; 允許右側合流拉框進料定點
      ANI     L4729  ; 右側合流拉框進料定點
      OUT     B1157  ; 右側合流拉框進料定點
6856  LD      B1157  ; 右側合流拉框進料定點
      OUT     B27E  ; 右側合流拉框進料定點SV
6858  LD      B1157  ; 右側合流拉框進料定點
      AND     SM412  ; 1.0 Sec Clock
      OR      L4729  ; 右側合流拉框進料定點
      OUT     M357  ; 右側合流拉框進料定點燈
6862  LD      L4027  ; 出料機構允許運轉
      ANDPI   M4139  ; 右側合流拉框夾爪異常
      OUT     L158  ; 允許右側合流拉框夾爪夾住
      OUT     L159  ; 允許右側合流拉框夾爪放開
6867  LD      L3653  ; 出料手動允許信號
      MPS
      AND     L158  ; 允許右側合流拉框夾爪夾住
      AND     M158  ; 右側合流拉框夾爪夾住SW
      OUT     T158 D106  ; 手動右側合流拉框夾爪夾住延遲
      MPP
      AND     L159  ; 允許右側合流拉框夾爪放開
      AND     M159  ; 右側合流拉框夾爪放開SW
      OUT     T159 D106  ; 手動右側合流拉框夾爪放開延遲
6882  LD      L3663  ; 出料自動允許信號
      MPS
      AND     L4732  ; 右側合流拉框夾爪有框
      AND     B26D  ; 右IR輸送變頻器INVB2運轉
      OUT     T471 K5  ; 右側合流拉框有框延遲
      MRD
      AND     L158  ; 允許右側合流拉框夾爪夾住
      AND     L4729  ; 右側合流拉框進料定點
      AND     L4735  ; 右側合流拉框昇降下定點
      AND     T471  ; 右側合流拉框有框延遲
      OUT     T458 D107  ; 自動右側合流拉框夾爪夾住延遲
      MPP
      AND     L159  ; 允許右側合流拉框夾爪放開
      AND     L4728  ; 右側合流拉框出料定點
      AND     L4735  ; 右側合流拉框昇降下定點
      OUT     T459 D107  ; 自動右側合流拉框夾爪放開延遲
